Staubli VAL3: Sychron_points.dtx

public jointRx jJointRx[1000]
  [0] = {j1=4.067745, j2=-15.879896, j3=110.159334, j4=0.000858, j5=81.483567, j6=22.610962}
  [1] = {j1=4.051625, j2=-15.882186, j3=110.160996, j4=0.002059, j5=81.484196, j6=22.594711}
  [2] = {j1=4.035504, j2=-15.884473, j3=110.162655, j4=0.00326, j5=81.484824, j6=22.578459}
  [3] = {j1=4.019382, j2=-15.886755, j3=110.164311, j4=0.004461, j5=81.485452, j6=22.562206}
  [4] = {j1=4.003258, j2=-15.889034, j3=110.165965, j4=0.005663, j5=81.486079, j6=22.545952}
  [5] = {j1=3.987134, j2=-15.89131, j3=110.167615, j4=0.006864, j5=81.486705, j6=22.529696}
  [6] = {j1=3.971008, j2=-15.893581, j3=110.169263, j4=0.008065, j5=81.487331, j6=22.51344}
  [7] = {j1=3.954882, j2=-15.895849, j3=110.170908, j4=0.009267, j5=81.487956, j6=22.497183}
  [8] = {j1=3.938754, j2=-15.898113, j3=110.17255, j4=0.010468, j5=81.48858, j6=22.480924}
  [9] = {j1=3.922625, j2=-15.900374, j3=110.17419, j4=0.01167, j5=81.489204, j6=22.464665}
  [10] = {j1=3.906496, j2=-15.90263, j3=110.175826, j4=0.012872, j5=81.489828, j6=22.448405}
  [11] = {j1=3.890365, j2=-15.904883, j3=110.17746, j4=0.014073, j5=81.49045, j6=22.432143}
  [12] = {j1=3.874233, j2=-15.907132, j3=110.179091, j4=0.015275, j5=81.491073, j6=22.415881}
  [13] = {j1=3.8581, j2=-15.909377, j3=110.180719, j4=0.016477, j5=81.491694, j6=22.399617}
  [14] = {j1=3.841966, j2=-15.911619, j3=110.182345, j4=0.017679, j5=81.492315, j6=22.383352}
  [15] = {j1=3.825831, j2=-15.913857, j3=110.183967, j4=0.018881, j5=81.492935, j6=22.367087}
  [16] = {j1=3.809695, j2=-15.916091, j3=110.185587, j4=0.020083, j5=81.493555, j6=22.35082}
  [17] = {j1=3.793558, j2=-15.918321, j3=110.187204, j4=0.021286, j5=81.494174, j6=22.334552}
  [18] = {j1=3.77742, j2=-15.920548, j3=110.188818, j4=0.022488, j5=81.494792, j6=22.318284}
  [19] = {j1=3.76128, j2=-15.922771, j3=110.190429, j4=0.02369, j5=81.49541, j6=22.302014}
  [20] = {j1=3.74514, j2=-15.92499, j3=110.192038, j4=0.024893, j5=81.496028, j6=22.285743}
  [21] = {j1=3.728999, j2=-15.927205, j3=110.193644, j4=0.026095, j5=81.496644, j6=22.269472}
  [22] = {j1=3.712857, j2=-15.929416, j3=110.195247, j4=0.027298, j5=81.49726, j6=22.253199}
  [23] = {j1=3.696713, j2=-15.931624, j3=110.196847, j4=0.028501, j5=81.497876, j6=22.236925}
  [24] = {j1=3.680569, j2=-15.933828, j3=110.198444, j4=0.029703, j5=81.49849, j6=22.22065}
  [25] = {j1=3.664424, j2=-15.936029, j3=110.200039, j4=0.030906, j5=81.499105, j6=22.204374}
  [26] = {j1=3.648277, j2=-15.938225, j3=110.20163, j4=0.032109, j5=81.499718, j6=22.188098}
  [27] = {j1=3.63213, j2=-15.940418, j3=110.203219, j4=0.033312, j5=81.500331, j6=22.17182}
  [28] = {j1=3.615981, j2=-15.942607, j3=110.204805, j4=0.034515, j5=81.500943, j6=22.155541}
  [29] = {j1=3.599832, j2=-15.944792, j3=110.206389, j4=0.035718, j5=81.501555, j6=22.139261}
  [30] = {j1=3.583681, j2=-15.946974, j3=110.207969, j4=0.036921, j5=81.502166, j6=22.12298}
  [31] = {j1=3.56753, j2=-15.949151, j3=110.209547, j4=0.038124, j5=81.502777, j6=22.106699}
  [32] = {j1=3.551377, j2=-15.951325, j3=110.211122, j4=0.039328, j5=81.503386, j6=22.090416}
  [33] = {j1=3.535224, j2=-15.953496, j3=110.212694, j4=0.040531, j5=81.503996, j6=22.074132}
  [34] = {j1=3.51907, j2=-15.955662, j3=110.214263, j4=0.041734, j5=81.504604, j6=22.057847}
  [35] = {j1=3.502914, j2=-15.957825, j3=110.21583, j4=0.042938, j5=81.505212, j6=22.041562}
  [36] = {j1=3.486758, j2=-15.959984, j3=110.217393, j4=0.044141, j5=81.50582, j6=22.025275}
  [37] = {j1=3.4706, j2=-15.962139, j3=110.218954, j4=0.045345, j5=81.506426, j6=22.008987}
  [38] = {j1=3.454442, j2=-15.96429, j3=110.220512, j4=0.046549, j5=81.507032, j6=21.992699}
  [39] = {j1=3.438282, j2=-15.966438, j3=110.222068, j4=0.047752, j5=81.507638, j6=21.976409}
  [40] = {j1=3.422122, j2=-15.968582, j3=110.22362, j4=0.048956, j5=81.508243, j6=21.960119}
  [41] = {j1=3.40596, j2=-15.970722, j3=110.22517, j4=0.05016, j5=81.508847, j6=21.943827}
  [42] = {j1=3.389798, j2=-15.972858, j3=110.226717, j4=0.051364, j5=81.509451, j6=21.927534}
  [43] = {j1=3.373635, j2=-15.97499, j3=110.228261, j4=0.052568, j5=81.510054, j6=21.911241}
  [44] = {j1=3.35747, j2=-15.977119, j3=110.229802, j4=0.053772, j5=81.510656, j6=21.894947}
  [45] = {j1=3.341305, j2=-15.979244, j3=110.23134, j4=0.054976, j5=81.511258, j6=21.878651}
  [46] = {j1=3.325139, j2=-15.981365, j3=110.232876, j4=0.056181, j5=81.511859, j6=21.862355}
  [47] = {j1=3.308971, j2=-15.983483, j3=110.234409, j4=0.057385, j5=81.512459, j6=21.846058}
  [48] = {j1=3.292803, j2=-15.985597, j3=110.235939, j4=0.058589, j5=81.513059, j6=21.829759}
  [49] = {j1=3.276634, j2=-15.987706, j3=110.237466, j4=0.059794, j5=81.513659, j6=21.81346}
  [50] = {j1=3.260464, j2=-15.989813, j3=110.23899, j4=0.060998, j5=81.514257, j6=21.79716}
  [51] = {j1=3.244293, j2=-15.991915, j3=110.240512, j4=0.062203, j5=81.514855, j6=21.780859}
  [52] = {j1=3.228121, j2=-15.994014, j3=110.242031, j4=0.063407, j5=81.515452, j6=21.764557}
  [53] = {j1=3.211948, j2=-15.996108, j3=110.243547, j4=0.064612, j5=81.516049, j6=21.748254}
  [54] = {j1=3.195774, j2=-15.998199, j3=110.24506, j4=0.065816, j5=81.516645, j6=21.73195}
  [55] = {j1=3.179599, j2=-16.000287, j3=110.24657, j4=0.067021, j5=81.517241, j6=21.715645}
  [56] = {j1=3.163423, j2=-16.00237, j3=110.248078, j4=0.068226, j5=81.517836, j6=21.699339}
  [57] = {j1=3.147246, j2=-16.00445, j3=110.249583, j4=0.069431, j5=81.51843, j6=21.683033}
  [58] = {j1=3.131068, j2=-16.006526, j3=110.251085, j4=0.070636, j5=81.519023, j6=21.666725}
  [59] = {j1=3.11489, j2=-16.008598, j3=110.252584, j4=0.071841, j5=81.519616, j6=21.650417}
  [60] = {j1=3.09871, j2=-16.010666, j3=110.25408, j4=0.073046, j5=81.520209, j6=21.634107}
  [61] = {j1=3.082529, j2=-16.012731, j3=110.255574, j4=0.074251, j5=81.5208, j6=21.617797}
  [62] = {j1=3.066348, j2=-16.014792, j3=110.257064, j4=0.075456, j5=81.521391, j6=21.601485}
  [63] = {j1=3.050165, j2=-16.016849, j3=110.258552, j4=0.076662, j5=81.521982, j6=21.585173}
  [64] = {j1=3.033982, j2=-16.018902, j3=110.260037, j4=0.077867, j5=81.522572, j6=21.56886}
  [65] = {j1=3.017798, j2=-16.020951, j3=110.26152, j4=0.079072, j5=81.523161, j6=21.552546}
  [66] = {j1=3.001613, j2=-16.022997, j3=110.262999, j4=0.080278, j5=81.523749, j6=21.536231}
  [67] = {j1=2.985426, j2=-16.025039, j3=110.264476, j4=0.081483, j5=81.524337, j6=21.519915}
  [68] = {j1=2.969239, j2=-16.027077, j3=110.26595, j4=0.082689, j5=81.524924, j6=21.503599}
  [69] = {j1=2.953051, j2=-16.029111, j3=110.267421, j4=0.083894, j5=81.525511, j6=21.487281}
  [70] = {j1=2.936863, j2=-16.031142, j3=110.268889, j4=0.0851, j5=81.526097, j6=21.470962}
  [71] = {j1=2.920673, j2=-16.033169, j3=110.270355, j4=0.086306, j5=81.526682, j6=21.454643}
  [72] = {j1=2.904482, j2=-16.035192, j3=110.271817, j4=0.087512, j5=81.527267, j6=21.438323}
  [73] = {j1=2.88829, j2=-16.037211, j3=110.273277, j4=0.088718, j5=81.527851, j6=21.422001}
  [74] = {j1=2.872098, j2=-16.039226, j3=110.274734, j4=0.089923, j5=81.528434, j6=21.405679}
  [75] = {j1=2.855905, j2=-16.041238, j3=110.276189, j4=0.091129, j5=81.529017, j6=21.389356}
  [76] = {j1=2.83971, j2=-16.043246, j3=110.27764, j4=0.092335, j5=81.529599, j6=21.373033}
  [77] = {j1=2.823515, j2=-16.04525, j3=110.279089, j4=0.093541, j5=81.53018, j6=21.356708}
  [78] = {j1=2.807319, j2=-16.04725, j3=110.280535, j4=0.094748, j5=81.530761, j6=21.340382}
  [79] = {j1=2.791122, j2=-16.049246, j3=110.281978, j4=0.095954, j5=81.531341, j6=21.324056}
  [80] = {j1=2.774924, j2=-16.051239, j3=110.283418, j4=0.09716, j5=81.531921, j6=21.307728}
  [81] = {j1=2.758725, j2=-16.053228, j3=110.284855, j4=0.098366, j5=81.5325, j6=21.2914}
  [82] = {j1=2.742526, j2=-16.055213, j3=110.28629, j4=0.099573, j5=81.533078, j6=21.275071}
  [83] = {j1=2.726325, j2=-16.057194, j3=110.287722, j4=0.100779, j5=81.533656, j6=21.258741}
  [84] = {j1=2.710124, j2=-16.059172, j3=110.289151, j4=0.101985, j5=81.534233, j6=21.24241}
  [85] = {j1=2.693922, j2=-16.061146, j3=110.290577, j4=0.103192, j5=81.534809, j6=21.226079}
  [86] = {j1=2.677718, j2=-16.063115, j3=110.292, j4=0.104399, j5=81.535385, j6=21.209746}
  [87] = {j1=2.661514, j2=-16.065082, j3=110.293421, j4=0.105605, j5=81.53596, j6=21.193413}
  [88] = {j1=2.645309, j2=-16.067044, j3=110.294839, j4=0.106812, j5=81.536534, j6=21.177078}
  [89] = {j1=2.629104, j2=-16.069002, j3=110.296253, j4=0.108019, j5=81.537108, j6=21.160743}
  [90] = {j1=2.612897, j2=-16.070957, j3=110.297666, j4=0.109225, j5=81.537681, j6=21.144407}
  [91] = {j1=2.59669, j2=-16.072908, j3=110.299075, j4=0.110432, j5=81.538253, j6=21.128071}
  [92] = {j1=2.580481, j2=-16.074855, j3=110.300481, j4=0.111639, j5=81.538825, j6=21.111733}
  [93] = {j1=2.564272, j2=-16.076798, j3=110.301885, j4=0.112846, j5=81.539396, j6=21.095394}
  [94] = {j1=2.548062, j2=-16.078738, j3=110.303286, j4=0.114053, j5=81.539967, j6=21.079055}
  [95] = {j1=2.531851, j2=-16.080674, j3=110.304684, j4=0.11526, j5=81.540537, j6=21.062715}
  [96] = {j1=2.515639, j2=-16.082606, j3=110.30608, j4=0.116467, j5=81.541106, j6=21.046374}
  [97] = {j1=2.499427, j2=-16.084534, j3=110.307472, j4=0.117674, j5=81.541674, j6=21.030032}
  [98] = {j1=2.483213, j2=-16.086458, j3=110.308862, j4=0.118881, j5=81.542242, j6=21.01369}
  [99] = {j1=2.466999, j2=-16.088378, j3=110.310249, j4=0.120089, j5=81.542809, j6=20.997346}
  [100] = {j1=2.450784, j2=-16.090295, j3=110.311633, j4=0.121296, j5=81.543376, j6=20.981002}
  [101] = {j1=2.434568, j2=-16.092208, j3=110.313014, j4=0.122503, j5=81.543942, j6=20.964657}
  [102] = {j1=2.418351, j2=-16.094117, j3=110.314392, j4=0.123711, j5=81.544507, j6=20.948311}
  [103] = {j1=2.402134, j2=-16.096023, j3=110.315768, j4=0.124918, j5=81.545072, j6=20.931964}
  [104] = {j1=2.385915, j2=-16.097924, j3=110.317141, j4=0.126126, j5=81.545636, j6=20.915617}
  [105] = {j1=2.369696, j2=-16.099822, j3=110.318511, j4=0.127333, j5=81.546199, j6=20.899268}
  [106] = {j1=2.353476, j2=-16.101716, j3=110.319878, j4=0.128541, j5=81.546762, j6=20.882919}
  [107] = {j1=2.337255, j2=-16.103606, j3=110.321243, j4=0.129748, j5=81.547324, j6=20.866569}
  [108] = {j1=2.321033, j2=-16.105492, j3=110.322604, j4=0.130956, j5=81.547885, j6=20.850218}
  [109] = {j1=2.304811, j2=-16.107374, j3=110.323963, j4=0.132164, j5=81.548446, j6=20.833867}
  [110] = {j1=2.288587, j2=-16.109253, j3=110.325319, j4=0.133371, j5=81.549006, j6=20.817514}
  [111] = {j1=2.272363, j2=-16.111128, j3=110.326672, j4=0.134579, j5=81.549565, j6=20.801161}
  [112] = {j1=2.256138, j2=-16.112999, j3=110.328023, j4=0.135787, j5=81.550124, j6=20.784807}
  [113] = {j1=2.239912, j2=-16.114866, j3=110.32937, j4=0.136995, j5=81.550682, j6=20.768453}
  [114] = {j1=2.223686, j2=-16.11673, j3=110.330715, j4=0.138203, j5=81.551239, j6=20.752097}
  [115] = {j1=2.207459, j2=-16.118589, j3=110.332057, j4=0.139411, j5=81.551796, j6=20.735741}
  [116] = {j1=2.19123, j2=-16.120445, j3=110.333396, j4=0.140619, j5=81.552352, j6=20.719384}
  [117] = {j1=2.175001, j2=-16.122297, j3=110.334732, j4=0.141827, j5=81.552907, j6=20.703026}
  [118] = {j1=2.158772, j2=-16.124145, j3=110.336066, j4=0.143035, j5=81.553462, j6=20.686667}
  [119] = {j1=2.142541, j2=-16.125989, j3=110.337397, j4=0.144243, j5=81.554016, j6=20.670308}
  [120] = {j1=2.12631, j2=-16.12783, j3=110.338725, j4=0.145452, j5=81.554569, j6=20.653948}
  [121] = {j1=2.110078, j2=-16.129667, j3=110.34005, j4=0.14666, j5=81.555122, j6=20.637587}
  [122] = {j1=2.093845, j2=-16.1315, j3=110.341372, j4=0.147868, j5=81.555674, j6=20.621225}
  [123] = {j1=2.077611, j2=-16.133329, j3=110.342692, j4=0.149076, j5=81.556226, j6=20.604862}
  [124] = {j1=2.061376, j2=-16.135154, j3=110.344008, j4=0.150285, j5=81.556776, j6=20.588499}
  [125] = {j1=2.045141, j2=-16.136975, j3=110.345322, j4=0.151493, j5=81.557327, j6=20.572135}
  [126] = {j1=2.028905, j2=-16.138793, j3=110.346633, j4=0.152702, j5=81.557876, j6=20.55577}
  [127] = {j1=2.012668, j2=-16.140607, j3=110.347941, j4=0.15391, j5=81.558425, j6=20.539405}
  [128] = {j1=1.996431, j2=-16.142417, j3=110.349247, j4=0.155119, j5=81.558973, j6=20.523038}
  [129] = {j1=1.980192, j2=-16.144223, j3=110.350549, j4=0.156327, j5=81.55952, j6=20.506671}
  [130] = {j1=1.963953, j2=-16.146026, j3=110.351849, j4=0.157536, j5=81.560067, j6=20.490304}
  [131] = {j1=1.947714, j2=-16.147824, j3=110.353146, j4=0.158745, j5=81.560613, j6=20.473935}
  [132] = {j1=1.931473, j2=-16.149619, j3=110.354441, j4=0.159954, j5=81.561159, j6=20.457566}
  [133] = {j1=1.915232, j2=-16.15141, j3=110.355732, j4=0.161162, j5=81.561703, j6=20.441196}
  [134] = {j1=1.898989, j2=-16.153197, j3=110.357021, j4=0.162371, j5=81.562247, j6=20.424825}
  [135] = {j1=1.882747, j2=-16.15498, j3=110.358306, j4=0.16358, j5=81.562791, j6=20.408454}
  [136] = {j1=1.866503, j2=-16.15676, j3=110.359589, j4=0.164789, j5=81.563334, j6=20.392081}
  [137] = {j1=1.850259, j2=-16.158535, j3=110.360869, j4=0.165998, j5=81.563876, j6=20.375708}
  [138] = {j1=1.834014, j2=-16.160307, j3=110.362147, j4=0.167207, j5=81.564417, j6=20.359335}
  [139] = {j1=1.817768, j2=-16.162075, j3=110.363421, j4=0.168416, j5=81.564958, j6=20.34296}
  [140] = {j1=1.801521, j2=-16.163839, j3=110.364693, j4=0.169625, j5=81.565498, j6=20.326585}
  [141] = {j1=1.785274, j2=-16.165599, j3=110.365962, j4=0.170834, j5=81.566037, j6=20.310209}
  [142] = {j1=1.769026, j2=-16.167356, j3=110.367228, j4=0.172043, j5=81.566576, j6=20.293833}
  [143] = {j1=1.752777, j2=-16.169109, j3=110.368492, j4=0.173252, j5=81.567114, j6=20.277455}
  [144] = {j1=1.736527, j2=-16.170857, j3=110.369752, j4=0.174461, j5=81.567651, j6=20.261077}
  [145] = {j1=1.720277, j2=-16.172602, j3=110.37101, j4=0.175671, j5=81.568188, j6=20.244699}
  [146] = {j1=1.704026, j2=-16.174344, j3=110.372265, j4=0.17688, j5=81.568724, j6=20.228319}
  [147] = {j1=1.687775, j2=-16.176081, j3=110.373517, j4=0.178089, j5=81.569259, j6=20.211939}
  [148] = {j1=1.671522, j2=-16.177815, j3=110.374766, j4=0.179298, j5=81.569794, j6=20.195558}
  [149] = {j1=1.655269, j2=-16.179544, j3=110.376012, j4=0.180508, j5=81.570328, j6=20.179177}
  [150] = {j1=1.639015, j2=-16.18127, j3=110.377256, j4=0.181717, j5=81.570861, j6=20.162795}
  [151] = {j1=1.622761, j2=-16.182992, j3=110.378497, j4=0.182927, j5=81.571394, j6=20.146412}
  [152] = {j1=1.606505, j2=-16.18471, j3=110.379735, j4=0.184136, j5=81.571926, j6=20.130028}
  [153] = {j1=1.59025, j2=-16.186425, j3=110.38097, j4=0.185346, j5=81.572457, j6=20.113644}
  [154] = {j1=1.573993, j2=-16.188135, j3=110.382203, j4=0.186555, j5=81.572988, j6=20.097259}
  [155] = {j1=1.557736, j2=-16.189842, j3=110.383432, j4=0.187765, j5=81.573518, j6=20.080873}
  [156] = {j1=1.541478, j2=-16.191545, j3=110.384659, j4=0.188974, j5=81.574047, j6=20.064487}
  [157] = {j1=1.525219, j2=-16.193244, j3=110.385883, j4=0.190184, j5=81.574576, j6=20.0481}
  [158] = {j1=1.508959, j2=-16.194939, j3=110.387104, j4=0.191394, j5=81.575104, j6=20.031712}
  [159] = {j1=1.492699, j2=-16.196631, j3=110.388322, j4=0.192603, j5=81.575631, j6=20.015324}
  [160] = {j1=1.476438, j2=-16.198318, j3=110.389538, j4=0.193813, j5=81.576157, j6=19.998935}
  [161] = {j1=1.460177, j2=-16.200002, j3=110.390751, j4=0.195023, j5=81.576683, j6=19.982545}
  [162] = {j1=1.443915, j2=-16.201682, j3=110.391961, j4=0.196233, j5=81.577209, j6=19.966155}
  [163] = {j1=1.427652, j2=-16.203358, j3=110.393168, j4=0.197443, j5=81.577733, j6=19.949764}
  [164] = {j1=1.411388, j2=-16.20503, j3=110.394372, j4=0.198653, j5=81.578257, j6=19.933372}
  [165] = {j1=1.395124, j2=-16.206698, j3=110.395574, j4=0.199862, j5=81.57878, j6=19.91698}
  [166] = {j1=1.378859, j2=-16.208363, j3=110.396772, j4=0.201072, j5=81.579302, j6=19.900586}
  [167] = {j1=1.362594, j2=-16.210024, j3=110.397968, j4=0.202282, j5=81.579824, j6=19.884193}
  [168] = {j1=1.346328, j2=-16.211681, j3=110.399161, j4=0.203492, j5=81.580345, j6=19.867798}
  [169] = {j1=1.330061, j2=-16.213334, j3=110.400352, j4=0.204702, j5=81.580866, j6=19.851403}
  [170] = {j1=1.313793, j2=-16.214983, j3=110.401539, j4=0.205912, j5=81.581385, j6=19.835008}
  [171] = {j1=1.297525, j2=-16.216628, j3=110.402724, j4=0.207123, j5=81.581904, j6=19.818612}
  [172] = {j1=1.281256, j2=-16.21827, j3=110.403905, j4=0.208333, j5=81.582423, j6=19.802215}
  [173] = {j1=1.264987, j2=-16.219907, j3=110.405085, j4=0.209543, j5=81.58294, j6=19.785817}
  [174] = {j1=1.248717, j2=-16.221541, j3=110.406261, j4=0.210753, j5=81.583457, j6=19.769419}
  [175] = {j1=1.232446, j2=-16.223171, j3=110.407434, j4=0.211963, j5=81.583974, j6=19.75302}
  [176] = {j1=1.216174, j2=-16.224797, j3=110.408605, j4=0.213173, j5=81.584489, j6=19.736621}
  [177] = {j1=1.199902, j2=-16.22642, j3=110.409772, j4=0.214384, j5=81.585004, j6=19.720221}
  [178] = {j1=1.183629, j2=-16.228038, j3=110.410937, j4=0.215594, j5=81.585518, j6=19.70382}
  [179] = {j1=1.167356, j2=-16.229653, j3=110.4121, j4=0.216804, j5=81.586032, j6=19.687418}
  [180] = {j1=1.151082, j2=-16.231263, j3=110.413259, j4=0.218015, j5=81.586545, j6=19.671017}
  [181] = {j1=1.134807, j2=-16.23287, j3=110.414416, j4=0.219225, j5=81.587057, j6=19.654614}
  [182] = {j1=1.118532, j2=-16.234473, j3=110.415569, j4=0.220435, j5=81.587568, j6=19.638211}
  [183] = {j1=1.102256, j2=-16.236073, j3=110.41672, j4=0.221646, j5=81.588079, j6=19.621807}
  [184] = {j1=1.08598, j2=-16.237668, j3=110.417868, j4=0.222856, j5=81.588589, j6=19.605402}
  [185] = {j1=1.069703, j2=-16.23926, j3=110.419014, j4=0.224067, j5=81.589099, j6=19.588997}
  [186] = {j1=1.053425, j2=-16.240847, j3=110.420156, j4=0.225277, j5=81.589607, j6=19.572592}
  [187] = {j1=1.037147, j2=-16.242431, j3=110.421296, j4=0.226488, j5=81.590115, j6=19.556186}
  [188] = {j1=1.020868, j2=-16.244011, j3=110.422433, j4=0.227698, j5=81.590623, j6=19.539779}
  [189] = {j1=1.004588, j2=-16.245587, j3=110.423567, j4=0.228909, j5=81.591129, j6=19.523371}
  [190] = {j1=0.988308, j2=-16.247159, j3=110.424698, j4=0.23012, j5=81.591635, j6=19.506963}
  [191] = {j1=0.972027, j2=-16.248728, j3=110.425826, j4=0.23133, j5=81.592141, j6=19.490555}
  [192] = {j1=0.955745, j2=-16.250292, j3=110.426952, j4=0.232541, j5=81.592645, j6=19.474145}
  [193] = {j1=0.939463, j2=-16.251853, j3=110.428075, j4=0.233752, j5=81.593149, j6=19.457736}
  [194] = {j1=0.923181, j2=-16.25341, j3=110.429195, j4=0.234962, j5=81.593652, j6=19.441325}
  [195] = {j1=0.906898, j2=-16.254963, j3=110.430312, j4=0.236173, j5=81.594155, j6=19.424914}
  [196] = {j1=0.890614, j2=-16.256512, j3=110.431426, j4=0.237384, j5=81.594656, j6=19.408503}
  [197] = {j1=0.874329, j2=-16.258058, j3=110.432538, j4=0.238594, j5=81.595157, j6=19.392091}
  [198] = {j1=0.858044, j2=-16.259599, j3=110.433647, j4=0.239805, j5=81.595658, j6=19.375678}
  [199] = {j1=0.841759, j2=-16.261137, j3=110.434753, j4=0.241016, j5=81.596157, j6=19.359265}
  [200] = {j1=0.825473, j2=-16.262671, j3=110.435856, j4=0.242227, j5=81.596656, j6=19.342851}
  [201] = {j1=0.809186, j2=-16.264201, j3=110.436956, j4=0.243438, j5=81.597155, j6=19.326436}
  [202] = {j1=0.792898, j2=-16.265727, j3=110.438054, j4=0.244649, j5=81.597652, j6=19.310021}
  [203] = {j1=0.77661, j2=-16.267249, j3=110.439148, j4=0.24586, j5=81.598149, j6=19.293606}
  [204] = {j1=0.760322, j2=-16.268767, j3=110.44024, j4=0.24707, j5=81.598645, j6=19.27719}
  [205] = {j1=0.744033, j2=-16.270282, j3=110.441329, j4=0.248281, j5=81.599141, j6=19.260773}
  [206] = {j1=0.727743, j2=-16.271792, j3=110.442415, j4=0.249492, j5=81.599636, j6=19.244356}
  [207] = {j1=0.711453, j2=-16.273299, j3=110.443499, j4=0.250703, j5=81.60013, j6=19.227938}
  [208] = {j1=0.695162, j2=-16.274802, j3=110.44458, j4=0.251914, j5=81.600623, j6=19.21152}
  [209] = {j1=0.678871, j2=-16.276301, j3=110.445657, j4=0.253125, j5=81.601116, j6=19.195101}
  [210] = {j1=0.662579, j2=-16.277796, j3=110.446732, j4=0.254336, j5=81.601608, j6=19.178681}
  [211] = {j1=0.646287, j2=-16.279288, j3=110.447805, j4=0.255547, j5=81.602099, j6=19.162261}
  [212] = {j1=0.629994, j2=-16.280775, j3=110.448874, j4=0.256758, j5=81.60259, j6=19.145841}
  [213] = {j1=0.6137, j2=-16.282259, j3=110.449941, j4=0.25797, j5=81.60308, j6=19.12942}
  [214] = {j1=0.597406, j2=-16.283739, j3=110.451004, j4=0.259181, j5=81.603569, j6=19.112998}
  [215] = {j1=0.581111, j2=-16.285214, j3=110.452065, j4=0.260392, j5=81.604057, j6=19.096576}
  [216] = {j1=0.564816, j2=-16.286687, j3=110.453123, j4=0.261603, j5=81.604545, j6=19.080153}
  [217] = {j1=0.548521, j2=-16.288155, j3=110.454179, j4=0.262814, j5=81.605032, j6=19.06373}
  [218] = {j1=0.532224, j2=-16.289619, j3=110.455231, j4=0.264025, j5=81.605518, j6=19.047307}
  [219] = {j1=0.515928, j2=-16.29108, j3=110.456281, j4=0.265236, j5=81.606004, j6=19.030882}
  [220] = {j1=0.49963, j2=-16.292536, j3=110.457328, j4=0.266448, j5=81.606489, j6=19.014458}
  [221] = {j1=0.483332, j2=-16.293989, j3=110.458372, j4=0.267659, j5=81.606973, j6=18.998032}
  [222] = {j1=0.467034, j2=-16.295438, j3=110.459413, j4=0.26887, j5=81.607457, j6=18.981607}
  [223] = {j1=0.450735, j2=-16.296883, j3=110.460452, j4=0.270081, j5=81.60794, j6=18.96518}
  [224] = {j1=0.434436, j2=-16.298324, j3=110.461487, j4=0.271293, j5=81.608422, j6=18.948753}
  [225] = {j1=0.418136, j2=-16.299761, j3=110.46252, j4=0.272504, j5=81.608903, j6=18.932326}
  [226] = {j1=0.401835, j2=-16.301195, j3=110.46355, j4=0.273715, j5=81.609384, j6=18.915898}
  [227] = {j1=0.385534, j2=-16.302624, j3=110.464578, j4=0.274926, j5=81.609864, j6=18.89947}
  [228] = {j1=0.369233, j2=-16.30405, j3=110.465602, j4=0.276138, j5=81.610343, j6=18.883041}
  [229] = {j1=0.352931, j2=-16.305472, j3=110.466624, j4=0.277349, j5=81.610822, j6=18.866612}
  [230] = {j1=0.336628, j2=-16.30689, j3=110.467642, j4=0.27856, j5=81.6113, j6=18.850182}
  [231] = {j1=0.320325, j2=-16.308304, j3=110.468658, j4=0.279772, j5=81.611777, j6=18.833752}
  [232] = {j1=0.304022, j2=-16.309714, j3=110.469671, j4=0.280983, j5=81.612253, j6=18.817321}
  [233] = {j1=0.287718, j2=-16.31112, j3=110.470682, j4=0.282195, j5=81.612729, j6=18.80089}
  [234] = {j1=0.271413, j2=-16.312523, j3=110.471689, j4=0.283406, j5=81.613204, j6=18.784458}
  [235] = {j1=0.255108, j2=-16.313921, j3=110.472694, j4=0.284617, j5=81.613678, j6=18.768026}
  [236] = {j1=0.238803, j2=-16.315316, j3=110.473696, j4=0.285829, j5=81.614152, j6=18.751593}
  [237] = {j1=0.222497, j2=-16.316707, j3=110.474695, j4=0.28704, j5=81.614625, j6=18.73516}
  [238] = {j1=0.20619, j2=-16.318094, j3=110.475691, j4=0.288252, j5=81.615097, j6=18.718726}
  [239] = {j1=0.189883, j2=-16.319477, j3=110.476685, j4=0.289463, j5=81.615569, j6=18.702292}
  [240] = {j1=0.173576, j2=-16.320856, j3=110.477676, j4=0.290675, j5=81.616039, j6=18.685858}
  [241] = {j1=0.157268, j2=-16.322232, j3=110.478663, j4=0.291886, j5=81.61651, j6=18.669423}
  [242] = {j1=0.14096, j2=-16.323603, j3=110.479648, j4=0.293097, j5=81.616979, j6=18.652987}
  [243] = {j1=0.124651, j2=-16.324971, j3=110.480631, j4=0.294309, j5=81.617447, j6=18.636551}
  [244] = {j1=0.108341, j2=-16.326335, j3=110.48161, j4=0.29552, j5=81.617915, j6=18.620115}
  [245] = {j1=0.092032, j2=-16.327695, j3=110.482587, j4=0.296732, j5=81.618383, j6=18.603678}
  [246] = {j1=0.075721, j2=-16.329051, j3=110.48356, j4=0.297943, j5=81.618849, j6=18.587241}
  [247] = {j1=0.059411, j2=-16.330403, j3=110.484531, j4=0.299155, j5=81.619315, j6=18.570803}
  [248] = {j1=0.043099, j2=-16.331751, j3=110.4855, j4=0.300367, j5=81.61978, j6=18.554364}
  [249] = {j1=0.026788, j2=-16.333096, j3=110.486465, j4=0.301578, j5=81.620244, j6=18.537926}
  [250] = {j1=0.010476, j2=-16.334436, j3=110.487427, j4=0.30279, j5=81.620708, j6=18.521487}
  [251] = {j1=-0.005837, j2=-16.335773, j3=110.488387, j4=0.304001, j5=81.621171, j6=18.505047}
  [252] = {j1=-0.02215, j2=-16.337106, j3=110.489344, j4=0.305213, j5=81.621633, j6=18.488607}
  [253] = {j1=-0.038463, j2=-16.338434, j3=110.490298, j4=0.306424, j5=81.622094, j6=18.472167}
  [254] = {j1=-0.054777, j2=-16.339759, j3=110.491249, j4=0.307636, j5=81.622555, j6=18.455726}
  [255] = {j1=-0.071092, j2=-16.341081, j3=110.492198, j4=0.308847, j5=81.623015, j6=18.439284}
  [256] = {j1=-0.087406, j2=-16.342398, j3=110.493144, j4=0.310059, j5=81.623475, j6=18.422843}
  [257] = {j1=-0.103722, j2=-16.343711, j3=110.494086, j4=0.311271, j5=81.623933, j6=18.406401}
  [258] = {j1=-0.120037, j2=-16.345021, j3=110.495026, j4=0.312482, j5=81.624391, j6=18.389958}
  [259] = {j1=-0.136353, j2=-16.346326, j3=110.495964, j4=0.313694, j5=81.624848, j6=18.373515}
  [260] = {j1=-0.15267, j2=-16.347628, j3=110.496898, j4=0.314905, j5=81.625305, j6=18.357072}
  [261] = {j1=-0.168987, j2=-16.348926, j3=110.49783, j4=0.316117, j5=81.62576, j6=18.340628}
  [262] = {j1=-0.185304, j2=-16.35022, j3=110.498758, j4=0.317329, j5=81.626215, j6=18.324184}
  [263] = {j1=-0.201622, j2=-16.35151, j3=110.499684, j4=0.31854, j5=81.62667, j6=18.307739}
  [264] = {j1=-0.21794, j2=-16.352796, j3=110.500608, j4=0.319752, j5=81.627123, j6=18.291294}
  [265] = {j1=-0.234259, j2=-16.354079, j3=110.501528, j4=0.320963, j5=81.627576, j6=18.274848}
  [266] = {j1=-0.250578, j2=-16.355357, j3=110.502445, j4=0.322175, j5=81.628028, j6=18.258403}
  [267] = {j1=-0.266897, j2=-16.356632, j3=110.50336, j4=0.323387, j5=81.62848, j6=18.241956}
  [268] = {j1=-0.283217, j2=-16.357903, j3=110.504272, j4=0.324598, j5=81.62893, j6=18.22551}
  [269] = {j1=-0.299537, j2=-16.359169, j3=110.505181, j4=0.32581, j5=81.62938, j6=18.209063}
  [270] = {j1=-0.315858, j2=-16.360432, j3=110.506087, j4=0.327022, j5=81.629829, j6=18.192615}
  [271] = {j1=-0.332179, j2=-16.361691, j3=110.506991, j4=0.328233, j5=81.630278, j6=18.176167}
  [272] = {j1=-0.3485, j2=-16.362947, j3=110.507892, j4=0.329445, j5=81.630726, j6=18.159719}
  [273] = {j1=-0.364822, j2=-16.364198, j3=110.508789, j4=0.330656, j5=81.631173, j6=18.143271}
  [274] = {j1=-0.381144, j2=-16.365445, j3=110.509684, j4=0.331868, j5=81.631619, j6=18.126822}
  [275] = {j1=-0.397467, j2=-16.366689, j3=110.510577, j4=0.33308, j5=81.632065, j6=18.110372}
  [276] = {j1=-0.41379, j2=-16.367928, j3=110.511466, j4=0.334291, j5=81.632509, j6=18.093923}
  [277] = {j1=-0.430113, j2=-16.369164, j3=110.512353, j4=0.335503, j5=81.632954, j6=18.077472}
  [278] = {j1=-0.446437, j2=-16.370396, j3=110.513236, j4=0.336715, j5=81.633397, j6=18.061022}
  [279] = {j1=-0.462761, j2=-16.371624, j3=110.514117, j4=0.337926, j5=81.63384, j6=18.044571}
  [280] = {j1=-0.479086, j2=-16.372848, j3=110.514996, j4=0.339138, j5=81.634282, j6=18.02812}
  [281] = {j1=-0.495411, j2=-16.374068, j3=110.515871, j4=0.340349, j5=81.634723, j6=18.011668}
  [282] = {j1=-0.511736, j2=-16.375285, j3=110.516743, j4=0.341561, j5=81.635163, j6=17.995217}
  [283] = {j1=-0.528062, j2=-16.376497, j3=110.517613, j4=0.342773, j5=81.635603, j6=17.978764}
  [284] = {j1=-0.544388, j2=-16.377706, j3=110.51848, j4=0.343984, j5=81.636042, j6=17.962312}
  [285] = {j1=-0.560714, j2=-16.37891, j3=110.519344, j4=0.345196, j5=81.636481, j6=17.945859}
  [286] = {j1=-0.577041, j2=-16.380111, j3=110.520205, j4=0.346408, j5=81.636918, j6=17.929405}
  [287] = {j1=-0.593368, j2=-16.381308, j3=110.521064, j4=0.347619, j5=81.637355, j6=17.912952}
  [288] = {j1=-0.609695, j2=-16.382501, j3=110.521919, j4=0.348831, j5=81.637791, j6=17.896498}
  [289] = {j1=-0.626023, j2=-16.38369, j3=110.522772, j4=0.350042, j5=81.638227, j6=17.880043}
  [290] = {j1=-0.642351, j2=-16.384875, j3=110.523622, j4=0.351254, j5=81.638661, j6=17.863589}
  [291] = {j1=-0.65868, j2=-16.386057, j3=110.524469, j4=0.352466, j5=81.639095, j6=17.847134}
  [292] = {j1=-0.675008, j2=-16.387234, j3=110.525314, j4=0.353677, j5=81.639528, j6=17.830678}
  [293] = {j1=-0.691338, j2=-16.388408, j3=110.526155, j4=0.354889, j5=81.639961, j6=17.814222}
  [294] = {j1=-0.707667, j2=-16.389577, j3=110.526994, j4=0.3561, j5=81.640393, j6=17.797766}
  [295] = {j1=-0.723997, j2=-16.390743, j3=110.52783, j4=0.357312, j5=81.640824, j6=17.78131}
  [296] = {j1=-0.740327, j2=-16.391905, j3=110.528663, j4=0.358523, j5=81.641254, j6=17.764853}
  [297] = {j1=-0.756658, j2=-16.393063, j3=110.529494, j4=0.359735, j5=81.641683, j6=17.748396}
  [298] = {j1=-0.772989, j2=-16.394217, j3=110.530321, j4=0.360947, j5=81.642112, j6=17.731939}
  [299] = {j1=-0.78932, j2=-16.395367, j3=110.531146, j4=0.362158, j5=81.64254, j6=17.715481}
  [300] = {j1=-0.805651, j2=-16.396513, j3=110.531968, j4=0.36337, j5=81.642968, j6=17.699023}
  [301] = {j1=-0.821983, j2=-16.397656, j3=110.532787, j4=0.364581, j5=81.643394, j6=17.682565}
  [302] = {j1=-0.838315, j2=-16.398794, j3=110.533603, j4=0.365793, j5=81.64382, j6=17.666107}
  [303] = {j1=-0.854648, j2=-16.399929, j3=110.534416, j4=0.367004, j5=81.644245, j6=17.649648}
  [304] = {j1=-0.87098, j2=-16.401059, j3=110.535227, j4=0.368216, j5=81.64467, j6=17.633189}
  [305] = {j1=-0.887314, j2=-16.402186, j3=110.536035, j4=0.369427, j5=81.645093, j6=17.616729}
  [306] = {j1=-0.903647, j2=-16.403309, j3=110.53684, j4=0.370639, j5=81.645516, j6=17.600269}
  [307] = {j1=-0.919981, j2=-16.404428, j3=110.537642, j4=0.37185, j5=81.645939, j6=17.583809}
  [308] = {j1=-0.936315, j2=-16.405543, j3=110.538441, j4=0.373062, j5=81.64636, j6=17.567349}
  [309] = {j1=-0.952649, j2=-16.406655, j3=110.539238, j4=0.374273, j5=81.646781, j6=17.550888}
  [310] = {j1=-0.968984, j2=-16.407762, j3=110.540032, j4=0.375485, j5=81.647201, j6=17.534427}
  [311] = {j1=-0.985318, j2=-16.408865, j3=110.540822, j4=0.376696, j5=81.64762, j6=17.517966}
  [312] = {j1=-1.001654, j2=-16.409965, j3=110.541611, j4=0.377907, j5=81.648039, j6=17.501505}
  [313] = {j1=-1.017989, j2=-16.41106, j3=110.542396, j4=0.379119, j5=81.648456, j6=17.485043}
  [314] = {j1=-1.034325, j2=-16.412152, j3=110.543178, j4=0.38033, j5=81.648873, j6=17.468581}
  [315] = {j1=-1.050661, j2=-16.41324, j3=110.543958, j4=0.381542, j5=81.64929, j6=17.452119}
  [316] = {j1=-1.066997, j2=-16.414324, j3=110.544735, j4=0.382753, j5=81.649705, j6=17.435656}
  [317] = {j1=-1.083334, j2=-16.415404, j3=110.545509, j4=0.383964, j5=81.65012, j6=17.419193}
  [318] = {j1=-1.099671, j2=-16.41648, j3=110.54628, j4=0.385176, j5=81.650534, j6=17.40273}
  [319] = {j1=-1.116008, j2=-16.417552, j3=110.547048, j4=0.386387, j5=81.650948, j6=17.386267}
  [320] = {j1=-1.132345, j2=-16.418621, j3=110.547814, j4=0.387598, j5=81.65136, j6=17.369803}
  [321] = {j1=-1.148683, j2=-16.419685, j3=110.548577, j4=0.38881, j5=81.651772, j6=17.353339}
  [322] = {j1=-1.165021, j2=-16.420746, j3=110.549337, j4=0.390021, j5=81.652183, j6=17.336875}
  [323] = {j1=-1.181359, j2=-16.421802, j3=110.550094, j4=0.391232, j5=81.652594, j6=17.32041}
  [324] = {j1=-1.197698, j2=-16.422855, j3=110.550848, j4=0.392444, j5=81.653003, j6=17.303946}
  [325] = {j1=-1.214036, j2=-16.423904, j3=110.5516, j4=0.393655, j5=81.653412, j6=17.287481}
  [326] = {j1=-1.230375, j2=-16.424949, j3=110.552348, j4=0.394866, j5=81.65382, j6=17.271016}
  [327] = {j1=-1.246715, j2=-16.42599, j3=110.553094, j4=0.396077, j5=81.654228, j6=17.25455}
  [328] = {j1=-1.263054, j2=-16.427027, j3=110.553837, j4=0.397289, j5=81.654634, j6=17.238085}
  [329] = {j1=-1.279394, j2=-16.42806, j3=110.554578, j4=0.3985, j5=81.65504, j6=17.221619}
  [330] = {j1=-1.295734, j2=-16.429089, j3=110.555315, j4=0.399711, j5=81.655445, j6=17.205153}
  [331] = {j1=-1.312074, j2=-16.430115, j3=110.55605, j4=0.400922, j5=81.65585, j6=17.188686}
  [332] = {j1=-1.328415, j2=-16.431136, j3=110.556782, j4=0.402133, j5=81.656254, j6=17.17222}
  [333] = {j1=-1.344755, j2=-16.432154, j3=110.557511, j4=0.403344, j5=81.656657, j6=17.155753}
  [334] = {j1=-1.361096, j2=-16.433168, j3=110.558237, j4=0.404556, j5=81.657059, j6=17.139286}
  [335] = {j1=-1.377437, j2=-16.434177, j3=110.55896, j4=0.405767, j5=81.65746, j6=17.122819}
  [336] = {j1=-1.393779, j2=-16.435183, j3=110.559681, j4=0.406978, j5=81.657861, j6=17.106351}
  [337] = {j1=-1.41012, j2=-16.436185, j3=110.560398, j4=0.408189, j5=81.658261, j6=17.089883}
  [338] = {j1=-1.426462, j2=-16.437183, j3=110.561113, j4=0.4094, j5=81.65866, j6=17.073416}
  [339] = {j1=-1.442804, j2=-16.438178, j3=110.561825, j4=0.410611, j5=81.659059, j6=17.056947}
  [340] = {j1=-1.459147, j2=-16.439168, j3=110.562535, j4=0.411822, j5=81.659456, j6=17.040479}
  [341] = {j1=-1.475489, j2=-16.440154, j3=110.563241, j4=0.413033, j5=81.659853, j6=17.024011}
  [342] = {j1=-1.491832, j2=-16.441137, j3=110.563945, j4=0.414244, j5=81.66025, j6=17.007542}
  [343] = {j1=-1.508175, j2=-16.442115, j3=110.564646, j4=0.415455, j5=81.660645, j6=16.991073}
  [344] = {j1=-1.524518, j2=-16.44309, j3=110.565344, j4=0.416666, j5=81.66104, j6=16.974604}
  [345] = {j1=-1.540861, j2=-16.44406, j3=110.566039, j4=0.417877, j5=81.661434, j6=16.958135}
  [346] = {j1=-1.557205, j2=-16.445027, j3=110.566731, j4=0.419088, j5=81.661827, j6=16.941665}
  [347] = {j1=-1.573549, j2=-16.44599, j3=110.567421, j4=0.420298, j5=81.66222, j6=16.925195}
  [348] = {j1=-1.589892, j2=-16.446949, j3=110.568108, j4=0.421509, j5=81.662611, j6=16.908725}
  [349] = {j1=-1.606237, j2=-16.447904, j3=110.568792, j4=0.42272, j5=81.663002, j6=16.892255}
  [350] = {j1=-1.622581, j2=-16.448855, j3=110.569473, j4=0.423931, j5=81.663393, j6=16.875785}
  [351] = {j1=-1.638925, j2=-16.449803, j3=110.570151, j4=0.425142, j5=81.663782, j6=16.859315}
  [352] = {j1=-1.65527, j2=-16.450746, j3=110.570827, j4=0.426352, j5=81.664171, j6=16.842844}
  [353] = {j1=-1.671615, j2=-16.451685, j3=110.571499, j4=0.427563, j5=81.664559, j6=16.826373}
  [354] = {j1=-1.68796, j2=-16.452621, j3=110.572169, j4=0.428774, j5=81.664946, j6=16.809902}
  [355] = {j1=-1.704305, j2=-16.453553, j3=110.572836, j4=0.429985, j5=81.665333, j6=16.793431}
  [356] = {j1=-1.720651, j2=-16.45448, j3=110.573501, j4=0.431195, j5=81.665719, j6=16.77696}
  [357] = {j1=-1.736996, j2=-16.455404, j3=110.574162, j4=0.432406, j5=81.666104, j6=16.760488}
  [358] = {j1=-1.753342, j2=-16.456324, j3=110.574821, j4=0.433617, j5=81.666488, j6=16.744017}
  [359] = {j1=-1.769688, j2=-16.45724, j3=110.575476, j4=0.434827, j5=81.666871, j6=16.727545}
  [360] = {j1=-1.786034, j2=-16.458152, j3=110.576129, j4=0.436038, j5=81.667254, j6=16.711073}
  [361] = {j1=-1.80238, j2=-16.45906, j3=110.57678, j4=0.437248, j5=81.667636, j6=16.694601}
  [362] = {j1=-1.818727, j2=-16.459964, j3=110.577427, j4=0.438459, j5=81.668017, j6=16.678129}
  [363] = {j1=-1.835073, j2=-16.460865, j3=110.578072, j4=0.439669, j5=81.668398, j6=16.661656}
  [364] = {j1=-1.85142, j2=-16.461761, j3=110.578713, j4=0.44088, j5=81.668778, j6=16.645184}
  [365] = {j1=-1.867767, j2=-16.462654, j3=110.579352, j4=0.44209, j5=81.669157, j6=16.628711}
  [366] = {j1=-1.884114, j2=-16.463542, j3=110.579988, j4=0.443301, j5=81.669535, j6=16.612238}
  [367] = {j1=-1.900461, j2=-16.464427, j3=110.580622, j4=0.444511, j5=81.669912, j6=16.595765}
  [368] = {j1=-1.900461, j2=-16.464427, j3=110.580622, j4=0.444511, j5=81.669912, j6=16.595765}
  [369] = {j1=-1.916822, j2=-16.465308, j3=110.581253, j4=0.445722, j5=81.670289, j6=16.579279}
  [370] = {j1=-1.933183, j2=-16.466186, j3=110.581881, j4=0.446933, j5=81.670666, j6=16.562793}
  [371] = {j1=-1.949544, j2=-16.467059, j3=110.582506, j4=0.448144, j5=81.671041, j6=16.546306}
  [372] = {j1=-1.965906, j2=-16.467929, j3=110.583129, j4=0.449354, j5=81.671416, j6=16.52982}
  [373] = {j1=-1.982267, j2=-16.468795, j3=110.583748, j4=0.450565, j5=81.67179, j6=16.513333}
  [374] = {j1=-1.998629, j2=-16.469657, j3=110.584365, j4=0.451776, j5=81.672163, j6=16.496846}
  [375] = {j1=-2.014991, j2=-16.470515, j3=110.584979, j4=0.452986, j5=81.672536, j6=16.480359}
  [376] = {j1=-2.031353, j2=-16.471369, j3=110.585591, j4=0.454197, j5=81.672908, j6=16.463872}
  [377] = {j1=-2.047715, j2=-16.472219, j3=110.586199, j4=0.455408, j5=81.673279, j6=16.447385}
  [378] = {j1=-2.064077, j2=-16.473065, j3=110.586805, j4=0.456618, j5=81.673649, j6=16.430898}
  [379] = {j1=-2.080439, j2=-16.473907, j3=110.587407, j4=0.457829, j5=81.674018, j6=16.41441}
  [380] = {j1=-2.096801, j2=-16.474746, j3=110.588007, j4=0.459039, j5=81.674387, j6=16.397923}
  [381] = {j1=-2.113164, j2=-16.47558, j3=110.588604, j4=0.46025, j5=81.674755, j6=16.381435}
  [382] = {j1=-2.129526, j2=-16.47641, j3=110.589199, j4=0.46146, j5=81.675122, j6=16.364947}
  [383] = {j1=-2.145889, j2=-16.477237, j3=110.58979, j4=0.462671, j5=81.675489, j6=16.348459}
  [384] = {j1=-2.162252, j2=-16.47806, j3=110.590379, j4=0.463881, j5=81.675854, j6=16.331971}
  [385] = {j1=-2.178615, j2=-16.478878, j3=110.590965, j4=0.465092, j5=81.676219, j6=16.315483}
  [386] = {j1=-2.194978, j2=-16.479693, j3=110.591548, j4=0.466302, j5=81.676583, j6=16.298995}
  [387] = {j1=-2.211341, j2=-16.480504, j3=110.592128, j4=0.467512, j5=81.676947, j6=16.282507}
  [388] = {j1=-2.227704, j2=-16.481311, j3=110.592705, j4=0.468723, j5=81.677309, j6=16.266018}
  [389] = {j1=-2.244067, j2=-16.482114, j3=110.59328, j4=0.469933, j5=81.677671, j6=16.24953}
  [390] = {j1=-2.260431, j2=-16.482913, j3=110.593852, j4=0.471143, j5=81.678032, j6=16.233041}
  [391] = {j1=-2.276794, j2=-16.483708, j3=110.594421, j4=0.472354, j5=81.678393, j6=16.216553}
  [392] = {j1=-2.293158, j2=-16.484499, j3=110.594987, j4=0.473564, j5=81.678752, j6=16.200064}
  [393] = {j1=-2.309521, j2=-16.485286, j3=110.59555, j4=0.474774, j5=81.679111, j6=16.183575}
  [394] = {j1=-2.325885, j2=-16.48607, j3=110.596111, j4=0.475984, j5=81.679469, j6=16.167086}
  [395] = {j1=-2.342249, j2=-16.486849, j3=110.596668, j4=0.477194, j5=81.679827, j6=16.150597}
  [396] = {j1=-2.358613, j2=-16.487625, j3=110.597223, j4=0.478405, j5=81.680183, j6=16.134108}
  [397] = {j1=-2.374977, j2=-16.488396, j3=110.597775, j4=0.479615, j5=81.680539, j6=16.117619}
  [398] = {j1=-2.391341, j2=-16.489164, j3=110.598324, j4=0.480825, j5=81.680894, j6=16.10113}
  [399] = {j1=-2.407705, j2=-16.489928, j3=110.598871, j4=0.482035, j5=81.681248, j6=16.084641}
  [400] = {j1=-2.424069, j2=-16.490687, j3=110.599414, j4=0.483245, j5=81.681602, j6=16.068152}
  [401] = {j1=-2.440433, j2=-16.491443, j3=110.599955, j4=0.484455, j5=81.681955, j6=16.051662}
  [402] = {j1=-2.456798, j2=-16.492195, j3=110.600493, j4=0.485665, j5=81.682307, j6=16.035173}
  [403] = {j1=-2.473162, j2=-16.492943, j3=110.601028, j4=0.486874, j5=81.682658, j6=16.018683}
  [404] = {j1=-2.489526, j2=-16.493687, j3=110.60156, j4=0.488084, j5=81.683008, j6=16.002194}
  [405] = {j1=-2.505891, j2=-16.494427, j3=110.60209, j4=0.489294, j5=81.683358, j6=15.985704}
  [406] = {j1=-2.522255, j2=-16.495164, j3=110.602616, j4=0.490504, j5=81.683707, j6=15.969215}
  [407] = {j1=-2.53862, j2=-16.495896, j3=110.60314, j4=0.491714, j5=81.684055, j6=15.952725}
  [408] = {j1=-2.554984, j2=-16.496624, j3=110.603661, j4=0.492923, j5=81.684402, j6=15.936235}
  [409] = {j1=-2.571349, j2=-16.497349, j3=110.604179, j4=0.494133, j5=81.684749, j6=15.919746}
  [410] = {j1=-2.587713, j2=-16.498069, j3=110.604695, j4=0.495343, j5=81.685095, j6=15.903256}
  [411] = {j1=-2.604078, j2=-16.498786, j3=110.605207, j4=0.496552, j5=81.68544, j6=15.886766}
  [412] = {j1=-2.620443, j2=-16.499498, j3=110.605717, j4=0.497762, j5=81.685784, j6=15.870276}
  [413] = {j1=-2.636808, j2=-16.500207, j3=110.606224, j4=0.498972, j5=81.686128, j6=15.853787}
  [414] = {j1=-2.653172, j2=-16.500912, j3=110.606728, j4=0.500181, j5=81.68647, j6=15.837297}
  [415] = {j1=-2.669537, j2=-16.501613, j3=110.607229, j4=0.501391, j5=81.686812, j6=15.820807}
  [416] = {j1=-2.685902, j2=-16.502309, j3=110.607728, j4=0.5026, j5=81.687154, j6=15.804317}
  [417] = {j1=-2.702267, j2=-16.503002, j3=110.608223, j4=0.503809, j5=81.687494, j6=15.787827}
  [418] = {j1=-2.718632, j2=-16.503691, j3=110.608716, j4=0.505019, j5=81.687834, j6=15.771337}
  [419] = {j1=-2.734996, j2=-16.504377, j3=110.609206, j4=0.506228, j5=81.688173, j6=15.754847}
  [420] = {j1=-2.751361, j2=-16.505058, j3=110.609693, j4=0.507437, j5=81.688511, j6=15.738357}
  [421] = {j1=-2.767726, j2=-16.505735, j3=110.610177, j4=0.508647, j5=81.688848, j6=15.721867}
  [422] = {j1=-2.784091, j2=-16.506408, j3=110.610659, j4=0.509856, j5=81.689185, j6=15.705377}
  [423] = {j1=-2.800456, j2=-16.507078, j3=110.611138, j4=0.511065, j5=81.689521, j6=15.688887}
  [424] = {j1=-2.816821, j2=-16.507743, j3=110.611613, j4=0.512274, j5=81.689856, j6=15.672397}
  [425] = {j1=-2.833186, j2=-16.508405, j3=110.612086, j4=0.513483, j5=81.69019, j6=15.655908}
  [426] = {j1=-2.84955, j2=-16.509062, j3=110.612557, j4=0.514693, j5=81.690524, j6=15.639418}
  [427] = {j1=-2.865915, j2=-16.509716, j3=110.613024, j4=0.515902, j5=81.690857, j6=15.622928}
  [428] = {j1=-2.88228, j2=-16.510365, j3=110.613489, j4=0.517111, j5=81.691189, j6=15.606438}
  [429] = {j1=-2.898645, j2=-16.511011, j3=110.61395, j4=0.51832, j5=81.69152, j6=15.589948}
  [430] = {j1=-2.91501, j2=-16.511653, j3=110.614409, j4=0.519528, j5=81.691851, j6=15.573458}
  [431] = {j1=-2.931375, j2=-16.512291, j3=110.614865, j4=0.520737, j5=81.69218, j6=15.556968}
  [432] = {j1=-2.947739, j2=-16.512925, j3=110.615319, j4=0.521946, j5=81.692509, j6=15.540478}
  [433] = {j1=-2.964104, j2=-16.513555, j3=110.615769, j4=0.523155, j5=81.692837, j6=15.523989}
  [434] = {j1=-2.980469, j2=-16.514181, j3=110.616217, j4=0.524364, j5=81.693165, j6=15.507499}
  [435] = {j1=-2.996834, j2=-16.514803, j3=110.616662, j4=0.525573, j5=81.693491, j6=15.491009}
  [436] = {j1=-3.013198, j2=-16.515421, j3=110.617104, j4=0.526781, j5=81.693817, j6=15.474519}
  [437] = {j1=-3.029563, j2=-16.516035, j3=110.617543, j4=0.52799, j5=81.694142, j6=15.45803}
  [438] = {j1=-3.045927, j2=-16.516646, j3=110.617979, j4=0.529198, j5=81.694467, j6=15.44154}
  [439] = {j1=-3.062292, j2=-16.517252, j3=110.618413, j4=0.530407, j5=81.69479, j6=15.42505}
  [440] = {j1=-3.078656, j2=-16.517855, j3=110.618844, j4=0.531616, j5=81.695113, j6=15.408561}
  [441] = {j1=-3.095021, j2=-16.518453, j3=110.619271, j4=0.532824, j5=81.695435, j6=15.392071}
  [442] = {j1=-3.111385, j2=-16.519048, j3=110.619697, j4=0.534032, j5=81.695756, j6=15.375582}
  [443] = {j1=-3.12775, j2=-16.519638, j3=110.620119, j4=0.535241, j5=81.696077, j6=15.359093}
  [444] = {j1=-3.144114, j2=-16.520225, j3=110.620538, j4=0.536449, j5=81.696396, j6=15.342603}
  [445] = {j1=-3.160478, j2=-16.520808, j3=110.620955, j4=0.537657, j5=81.696715, j6=15.326114}
  [446] = {j1=-3.176842, j2=-16.521387, j3=110.621369, j4=0.538866, j5=81.697033, j6=15.309625}
  [447] = {j1=-3.193207, j2=-16.521962, j3=110.62178, j4=0.540074, j5=81.697351, j6=15.293136}
  [448] = {j1=-3.209571, j2=-16.522532, j3=110.622188, j4=0.541282, j5=81.697667, j6=15.276647}
  [449] = {j1=-3.225935, j2=-16.523099, j3=110.622593, j4=0.54249, j5=81.697983, j6=15.260158}
  [450] = {j1=-3.242299, j2=-16.523663, j3=110.622996, j4=0.543698, j5=81.698298, j6=15.243669}
  [451] = {j1=-3.258662, j2=-16.524222, j3=110.623395, j4=0.544906, j5=81.698612, j6=15.22718}
  [452] = {j1=-3.275026, j2=-16.524777, j3=110.623792, j4=0.546114, j5=81.698926, j6=15.210691}
  [453] = {j1=-3.29139, j2=-16.525328, j3=110.624186, j4=0.547322, j5=81.699239, j6=15.194202}
  [454] = {j1=-3.307753, j2=-16.525875, j3=110.624577, j4=0.54853, j5=81.69955, j6=15.177714}
  [455] = {j1=-3.324117, j2=-16.526419, j3=110.624966, j4=0.549738, j5=81.699862, j6=15.161225}
  [456] = {j1=-3.34048, j2=-16.526958, j3=110.625351, j4=0.550946, j5=81.700172, j6=15.144737}
  [457] = {j1=-3.356844, j2=-16.527494, j3=110.625734, j4=0.552154, j5=81.700482, j6=15.128248}
  [458] = {j1=-3.373207, j2=-16.528025, j3=110.626114, j4=0.553361, j5=81.70079, j6=15.11176}
  [459] = {j1=-3.38957, j2=-16.528553, j3=110.626491, j4=0.554569, j5=81.701098, j6=15.095272}
  [460] = {j1=-3.405933, j2=-16.529077, j3=110.626866, j4=0.555776, j5=81.701406, j6=15.078784}
  [461] = {j1=-3.422296, j2=-16.529596, j3=110.627237, j4=0.556984, j5=81.701712, j6=15.062296}
  [462] = {j1=-3.438659, j2=-16.530112, j3=110.627606, j4=0.558192, j5=81.702018, j6=15.045808}
  [463] = {j1=-3.455022, j2=-16.530624, j3=110.627972, j4=0.559399, j5=81.702323, j6=15.02932}
  [464] = {j1=-3.471385, j2=-16.531132, j3=110.628335, j4=0.560606, j5=81.702627, j6=15.012832}
  [465] = {j1=-3.487747, j2=-16.531636, j3=110.628695, j4=0.561814, j5=81.70293, j6=14.996345}
  [466] = {j1=-3.50411, j2=-16.532136, j3=110.629052, j4=0.563021, j5=81.703233, j6=14.979857}
  [467] = {j1=-3.520472, j2=-16.532632, j3=110.629407, j4=0.564228, j5=81.703535, j6=14.96337}
  [468] = {j1=-3.536834, j2=-16.533124, j3=110.629758, j4=0.565436, j5=81.703836, j6=14.946883}
  [469] = {j1=-3.553196, j2=-16.533612, j3=110.630107, j4=0.566643, j5=81.704136, j6=14.930396}
  [470] = {j1=-3.569558, j2=-16.534096, j3=110.630453, j4=0.56785, j5=81.704436, j6=14.913909}
  [471] = {j1=-3.58592, j2=-16.534577, j3=110.630797, j4=0.569057, j5=81.704734, j6=14.897422}
  [472] = {j1=-3.602282, j2=-16.535053, j3=110.631137, j4=0.570264, j5=81.705032, j6=14.880935}
  [473] = {j1=-3.618643, j2=-16.535526, j3=110.631475, j4=0.571471, j5=81.70533, j6=14.864449}
  [474] = {j1=-3.635005, j2=-16.535994, j3=110.63181, j4=0.572678, j5=81.705626, j6=14.847962}
  [475] = {j1=-3.651366, j2=-16.536459, j3=110.632141, j4=0.573885, j5=81.705922, j6=14.831476}
  [476] = {j1=-3.667727, j2=-16.536919, j3=110.632471, j4=0.575091, j5=81.706216, j6=14.81499}
  [477] = {j1=-3.684088, j2=-16.537376, j3=110.632797, j4=0.576298, j5=81.70651, j6=14.798504}
  [478] = {j1=-3.700449, j2=-16.537829, j3=110.63312, j4=0.577505, j5=81.706804, j6=14.782018}
  [479] = {j1=-3.71681, j2=-16.538277, j3=110.633441, j4=0.578711, j5=81.707096, j6=14.765532}
  [480] = {j1=-3.733171, j2=-16.538722, j3=110.633759, j4=0.579918, j5=81.707388, j6=14.749047}
  [481] = {j1=-3.749531, j2=-16.539163, j3=110.634074, j4=0.581125, j5=81.707679, j6=14.732561}
  [482] = {j1=-3.765891, j2=-16.5396, j3=110.634386, j4=0.582331, j5=81.707969, j6=14.716076}
  [483] = {j1=-3.782251, j2=-16.540033, j3=110.634696, j4=0.583537, j5=81.708258, j6=14.699591}
  [484] = {j1=-3.798611, j2=-16.540462, j3=110.635002, j4=0.584744, j5=81.708547, j6=14.683106}
  [485] = {j1=-3.814971, j2=-16.540887, j3=110.635306, j4=0.58595, j5=81.708835, j6=14.666621}
  [486] = {j1=-3.831331, j2=-16.541308, j3=110.635607, j4=0.587156, j5=81.709122, j6=14.650137}
  [487] = {j1=-3.84769, j2=-16.541725, j3=110.635905, j4=0.588363, j5=81.709408, j6=14.633652}
  [488] = {j1=-3.86405, j2=-16.542139, j3=110.6362, j4=0.589569, j5=81.709693, j6=14.617168}
  [489] = {j1=-3.880409, j2=-16.542548, j3=110.636493, j4=0.590775, j5=81.709978, j6=14.600684}
  [490] = {j1=-3.896768, j2=-16.542953, j3=110.636783, j4=0.591981, j5=81.710262, j6=14.5842}
  [491] = {j1=-3.913126, j2=-16.543355, j3=110.637069, j4=0.593187, j5=81.710545, j6=14.567716}
  [492] = {j1=-3.929485, j2=-16.543752, j3=110.637353, j4=0.594393, j5=81.710827, j6=14.551233}
  [493] = {j1=-3.945843, j2=-16.544146, j3=110.637635, j4=0.595599, j5=81.711109, j6=14.534749}
  [494] = {j1=-3.962202, j2=-16.544536, j3=110.637913, j4=0.596804, j5=81.71139, j6=14.518266}
  [495] = {j1=-3.97856, j2=-16.544921, j3=110.638189, j4=0.59801, j5=81.71167, j6=14.501783}
  [496] = {j1=-3.994917, j2=-16.545303, j3=110.638461, j4=0.599216, j5=81.711949, j6=14.4853}
  [497] = {j1=-4.011275, j2=-16.545681, j3=110.638731, j4=0.600421, j5=81.712227, j6=14.468818}
  [498] = {j1=-4.027633, j2=-16.546054, j3=110.638998, j4=0.601627, j5=81.712505, j6=14.452335}
  [499] = {j1=-4.04399, j2=-16.546424, j3=110.639262, j4=0.602832, j5=81.712782, j6=14.435853}
  [500] = {j1=-4.060347, j2=-16.54679, j3=110.639524, j4=0.604038, j5=81.713058, j6=14.419371}
  [501] = {j1=-4.076704, j2=-16.547152, j3=110.639783, j4=0.605243, j5=81.713333, j6=14.402889}
  [502] = {j1=-4.09306, j2=-16.54751, j3=110.640038, j4=0.606449, j5=81.713608, j6=14.386408}
  [503] = {j1=-4.109417, j2=-16.547864, j3=110.640291, j4=0.607654, j5=81.713881, j6=14.369926}
  [504] = {j1=-4.125773, j2=-16.548214, j3=110.640541, j4=0.608859, j5=81.714154, j6=14.353445}
  [505] = {j1=-4.142129, j2=-16.548561, j3=110.640789, j4=0.610064, j5=81.714426, j6=14.336964}
  [506] = {j1=-4.158485, j2=-16.548903, j3=110.641033, j4=0.611269, j5=81.714698, j6=14.320483}
  [507] = {j1=-4.17484, j2=-16.549241, j3=110.641275, j4=0.612474, j5=81.714968, j6=14.304003}
  [508] = {j1=-4.191195, j2=-16.549576, j3=110.641514, j4=0.613679, j5=81.715238, j6=14.287523}
  [509] = {j1=-4.20755, j2=-16.549906, j3=110.64175, j4=0.614884, j5=81.715507, j6=14.271043}
  [510] = {j1=-4.223905, j2=-16.550232, j3=110.641983, j4=0.616089, j5=81.715775, j6=14.254563}
  [511] = {j1=-4.24026, j2=-16.550555, j3=110.642214, j4=0.617294, j5=81.716043, j6=14.238083}
  [512] = {j1=-4.256614, j2=-16.550873, j3=110.642441, j4=0.618498, j5=81.716309, j6=14.221604}
  [513] = {j1=-4.272968, j2=-16.551188, j3=110.642666, j4=0.619703, j5=81.716575, j6=14.205125}
  [514] = {j1=-4.289322, j2=-16.551499, j3=110.642888, j4=0.620908, j5=81.71684, j6=14.188646}
  [515] = {j1=-4.305676, j2=-16.551805, j3=110.643107, j4=0.622112, j5=81.717105, j6=14.172167}
  [516] = {j1=-4.322029, j2=-16.552108, j3=110.643323, j4=0.623317, j5=81.717368, j6=14.155689}
  [517] = {j1=-4.338383, j2=-16.552407, j3=110.643537, j4=0.624521, j5=81.717631, j6=14.139211}
  [518] = {j1=-4.354736, j2=-16.552702, j3=110.643747, j4=0.625725, j5=81.717893, j6=14.122733}
  [519] = {j1=-4.371088, j2=-16.552993, j3=110.643955, j4=0.62693, j5=81.718154, j6=14.106255}
  [520] = {j1=-4.387441, j2=-16.55328, j3=110.64416, j4=0.628134, j5=81.718414, j6=14.089778}
  [521] = {j1=-4.403793, j2=-16.553563, j3=110.644362, j4=0.629338, j5=81.718674, j6=14.073301}
  [522] = {j1=-4.420145, j2=-16.553842, j3=110.644562, j4=0.630542, j5=81.718933, j6=14.056824}
  [523] = {j1=-4.436496, j2=-16.554117, j3=110.644758, j4=0.631746, j5=81.719191, j6=14.040347}
  [524] = {j1=-4.452848, j2=-16.554388, j3=110.644952, j4=0.63295, j5=81.719448, j6=14.023871}
  [525] = {j1=-4.469199, j2=-16.554655, j3=110.645143, j4=0.634154, j5=81.719704, j6=14.007395}
  [526] = {j1=-4.485549, j2=-16.554919, j3=110.645331, j4=0.635357, j5=81.71996, j6=13.990919}
  [527] = {j1=-4.5019, j2=-16.555178, j3=110.645516, j4=0.636561, j5=81.720215, j6=13.974444}
  [528] = {j1=-4.51825, j2=-16.555433, j3=110.645699, j4=0.637765, j5=81.720469, j6=13.957968}
  [529] = {j1=-4.5346, j2=-16.555685, j3=110.645878, j4=0.638968, j5=81.720722, j6=13.941493}
  [530] = {j1=-4.55095, j2=-16.555932, j3=110.646055, j4=0.640172, j5=81.720975, j6=13.925019}
  [531] = {j1=-4.567299, j2=-16.556176, j3=110.646229, j4=0.641375, j5=81.721226, j6=13.908544}
  [532] = {j1=-4.583648, j2=-16.556416, j3=110.6464, j4=0.642579, j5=81.721477, j6=13.89207}
  [533] = {j1=-4.599997, j2=-16.556651, j3=110.646568, j4=0.643782, j5=81.721727, j6=13.875596}
  [534] = {j1=-4.616346, j2=-16.556883, j3=110.646734, j4=0.644985, j5=81.721977, j6=13.859123}
  [535] = {j1=-4.632694, j2=-16.557111, j3=110.646896, j4=0.646189, j5=81.722225, j6=13.84265}
  [536] = {j1=-4.649042, j2=-16.557334, j3=110.647056, j4=0.647392, j5=81.722473, j6=13.826177}
  [537] = {j1=-4.66539, j2=-16.557554, j3=110.647213, j4=0.648595, j5=81.72272, j6=13.809704}
  [538] = {j1=-4.681737, j2=-16.55777, j3=110.647368, j4=0.649798, j5=81.722966, j6=13.793232}
  [539] = {j1=-4.698084, j2=-16.557982, j3=110.647519, j4=0.651, j5=81.723212, j6=13.77676}
  [540] = {j1=-4.714431, j2=-16.55819, j3=110.647668, j4=0.652203, j5=81.723456, j6=13.760288}
  [541] = {j1=-4.730777, j2=-16.558394, j3=110.647813, j4=0.653406, j5=81.7237, j6=13.743817}
  [542] = {j1=-4.747123, j2=-16.558594, j3=110.647956, j4=0.654609, j5=81.723943, j6=13.727346}
  [543] = {j1=-4.763469, j2=-16.55879, j3=110.648096, j4=0.655811, j5=81.724185, j6=13.710875}
  [544] = {j1=-4.779814, j2=-16.558983, j3=110.648234, j4=0.657014, j5=81.724427, j6=13.694405}
  [545] = {j1=-4.796159, j2=-16.559171, j3=110.648368, j4=0.658216, j5=81.724667, j6=13.677934}
  [546] = {j1=-4.812504, j2=-16.559355, j3=110.6485, j4=0.659419, j5=81.724907, j6=13.661465}
  [547] = {j1=-4.828849, j2=-16.559535, j3=110.648628, j4=0.660621, j5=81.725146, j6=13.644995}
  [548] = {j1=-4.845193, j2=-16.559712, j3=110.648754, j4=0.661823, j5=81.725385, j6=13.628526}
  [549] = {j1=-4.861536, j2=-16.559884, j3=110.648878, j4=0.663025, j5=81.725622, j6=13.612057}
  [550] = {j1=-4.87788, j2=-16.560053, j3=110.648998, j4=0.664228, j5=81.725859, j6=13.595589}
  [551] = {j1=-4.894223, j2=-16.560217, j3=110.649115, j4=0.66543, j5=81.726095, j6=13.579121}
  [552] = {j1=-4.910566, j2=-16.560378, j3=110.64923, j4=0.666632, j5=81.72633, j6=13.562653}
  [553] = {j1=-4.926908, j2=-16.560535, j3=110.649342, j4=0.667833, j5=81.726564, j6=13.546185}
  [554] = {j1=-4.94325, j2=-16.560687, j3=110.649451, j4=0.669035, j5=81.726798, j6=13.529718}
  [555] = {j1=-4.959592, j2=-16.560836, j3=110.649557, j4=0.670237, j5=81.727031, j6=13.513252}
  [556] = {j1=-4.975933, j2=-16.560981, j3=110.649661, j4=0.671439, j5=81.727262, j6=13.496785}
  [557] = {j1=-4.992274, j2=-16.561122, j3=110.649761, j4=0.67264, j5=81.727494, j6=13.480319}
  [558] = {j1=-5.008615, j2=-16.561258, j3=110.649859, j4=0.673842, j5=81.727724, j6=13.463853}
  [559] = {j1=-5.024955, j2=-16.561391, j3=110.649954, j4=0.675043, j5=81.727954, j6=13.447388}
  [560] = {j1=-5.041295, j2=-16.56152, j3=110.650046, j4=0.676244, j5=81.728182, j6=13.430923}
  [561] = {j1=-5.057635, j2=-16.561645, j3=110.650135, j4=0.677446, j5=81.72841, j6=13.414459}
  [562] = {j1=-5.073974, j2=-16.561766, j3=110.650222, j4=0.678647, j5=81.728638, j6=13.397994}
  [563] = {j1=-5.090313, j2=-16.561884, j3=110.650306, j4=0.679848, j5=81.728864, j6=13.381531}
  [564] = {j1=-5.106651, j2=-16.561997, j3=110.650386, j4=0.681049, j5=81.72909, j6=13.365067}
  [565] = {j1=-5.12299, j2=-16.562106, j3=110.650464, j4=0.68225, j5=81.729315, j6=13.348604}
  [566] = {j1=-5.139327, j2=-16.562211, j3=110.65054, j4=0.683451, j5=81.729539, j6=13.332141}
  [567] = {j1=-5.155665, j2=-16.562313, j3=110.650612, j4=0.684652, j5=81.729762, j6=13.315679}
  [568] = {j1=-5.172002, j2=-16.56241, j3=110.650681, j4=0.685852, j5=81.729984, j6=13.299217}
  [569] = {j1=-5.188338, j2=-16.562503, j3=110.650748, j4=0.687053, j5=81.730206, j6=13.282755}
  [570] = {j1=-5.204674, j2=-16.562593, j3=110.650812, j4=0.688253, j5=81.730427, j6=13.266294}
  [571] = {j1=-5.22101, j2=-16.562678, j3=110.650873, j4=0.689454, j5=81.730647, j6=13.249833}
  [572] = {j1=-5.237345, j2=-16.56276, j3=110.650931, j4=0.690654, j5=81.730866, j6=13.233373}
  [573] = {j1=-5.25368, j2=-16.562838, j3=110.650987, j4=0.691855, j5=81.731085, j6=13.216913}
  [574] = {j1=-5.270015, j2=-16.562911, j3=110.651039, j4=0.693055, j5=81.731303, j6=13.200453}
  [575] = {j1=-5.286349, j2=-16.562981, j3=110.651089, j4=0.694255, j5=81.731519, j6=13.183994}
  [576] = {j1=-5.302683, j2=-16.563047, j3=110.651136, j4=0.695455, j5=81.731736, j6=13.167535}
  [577] = {j1=-5.319016, j2=-16.563109, j3=110.65118, j4=0.696655, j5=81.731951, j6=13.151077}
  [578] = {j1=-5.335349, j2=-16.563166, j3=110.651222, j4=0.697855, j5=81.732165, j6=13.134619}
  [579] = {j1=-5.351682, j2=-16.56322, j3=110.65126, j4=0.699055, j5=81.732379, j6=13.118161}
  [580] = {j1=-5.368014, j2=-16.56327, j3=110.651296, j4=0.700255, j5=81.732592, j6=13.101704}
  [581] = {j1=-5.384346, j2=-16.563316, j3=110.651329, j4=0.701454, j5=81.732804, j6=13.085247}
  [582] = {j1=-5.400677, j2=-16.563358, j3=110.651359, j4=0.702654, j5=81.733016, j6=13.068791}
  [583] = {j1=-5.417008, j2=-16.563397, j3=110.651386, j4=0.703853, j5=81.733226, j6=13.052335}
  [584] = {j1=-5.433338, j2=-16.563431, j3=110.65141, j4=0.705053, j5=81.733436, j6=13.035879}
  [585] = {j1=-5.449668, j2=-16.563461, j3=110.651432, j4=0.706252, j5=81.733645, j6=13.019424}
  [586] = {j1=-5.465998, j2=-16.563487, j3=110.651451, j4=0.707451, j5=81.733853, j6=13.00297}
  [587] = {j1=-5.482327, j2=-16.563509, j3=110.651467, j4=0.70865, j5=81.734061, j6=12.986516}
  [588] = {j1=-5.498655, j2=-16.563528, j3=110.65148, j4=0.70985, j5=81.734267, j6=12.970062}
  [589] = {j1=-5.514984, j2=-16.563542, j3=110.65149, j4=0.711049, j5=81.734473, j6=12.953608}
  [590] = {j1=-5.531311, j2=-16.563553, j3=110.651497, j4=0.712247, j5=81.734678, j6=12.937156}
  [591] = {j1=-5.547639, j2=-16.563559, j3=110.651502, j4=0.713446, j5=81.734882, j6=12.920703}
  [592] = {j1=-5.563966, j2=-16.563562, j3=110.651504, j4=0.714645, j5=81.735086, j6=12.904251}
  [593] = {j1=-5.580292, j2=-16.56356, j3=110.651503, j4=0.715844, j5=81.735288, j6=12.8878}
  [594] = {j1=-5.596618, j2=-16.563555, j3=110.651499, j4=0.717042, j5=81.73549, j6=12.871348}
  [595] = {j1=-5.612944, j2=-16.563546, j3=110.651492, j4=0.718241, j5=81.735691, j6=12.854898}
  [596] = {j1=-5.629269, j2=-16.563532, j3=110.651483, j4=0.719439, j5=81.735892, j6=12.838448}
  [597] = {j1=-5.645593, j2=-16.563515, j3=110.651471, j4=0.720637, j5=81.736091, j6=12.821998}
  [598] = {j1=-5.661918, j2=-16.563494, j3=110.651455, j4=0.721836, j5=81.73629, j6=12.805549}
  [599] = {j1=-5.678241, j2=-16.563469, j3=110.651437, j4=0.723034, j5=81.736487, j6=12.7891}
  [600] = {j1=-5.694565, j2=-16.56344, j3=110.651417, j4=0.724232, j5=81.736685, j6=12.772651}
  [601] = {j1=-5.710887, j2=-16.563407, j3=110.651393, j4=0.72543, j5=81.736881, j6=12.756204}
  [602] = {j1=-5.72721, j2=-16.56337, j3=110.651367, j4=0.726628, j5=81.737076, j6=12.739756}
  [603] = {j1=-5.743531, j2=-16.563329, j3=110.651337, j4=0.727825, j5=81.737271, j6=12.723309}
  [604] = {j1=-5.759853, j2=-16.563284, j3=110.651305, j4=0.729023, j5=81.737465, j6=12.706863}
  [605] = {j1=-5.776174, j2=-16.563235, j3=110.651271, j4=0.730221, j5=81.737658, j6=12.690417}
  [606] = {j1=-5.792494, j2=-16.563182, j3=110.651233, j4=0.731418, j5=81.73785, j6=12.673971}
  [607] = {j1=-5.808814, j2=-16.563126, j3=110.651192, j4=0.732616, j5=81.738042, j6=12.657526}
  [608] = {j1=-5.825133, j2=-16.563065, j3=110.651149, j4=0.733813, j5=81.738233, j6=12.641082}
  [609] = {j1=-5.841452, j2=-16.563, j3=110.651103, j4=0.73501, j5=81.738422, j6=12.624638}
  [610] = {j1=-5.85777, j2=-16.562932, j3=110.651054, j4=0.736207, j5=81.738612, j6=12.608194}
  [611] = {j1=-5.874088, j2=-16.562859, j3=110.651002, j4=0.737404, j5=81.7388, j6=12.591751}
  [612] = {j1=-5.890406, j2=-16.562783, j3=110.650947, j4=0.738601, j5=81.738987, j6=12.575309}
  [613] = {j1=-5.906723, j2=-16.562702, j3=110.65089, j4=0.739798, j5=81.739174, j6=12.558867}
  [614] = {j1=-5.923039, j2=-16.562618, j3=110.65083, j4=0.740995, j5=81.73936, j6=12.542425}
  [615] = {j1=-5.939355, j2=-16.562529, j3=110.650767, j4=0.742192, j5=81.739545, j6=12.525984}
  [616] = {j1=-5.95567, j2=-16.562437, j3=110.650701, j4=0.743388, j5=81.73973, j6=12.509544}
  [617] = {j1=-5.971985, j2=-16.562341, j3=110.650632, j4=0.744585, j5=81.739913, j6=12.493104}
  [618] = {j1=-5.988299, j2=-16.562241, j3=110.65056, j4=0.745781, j5=81.740096, j6=12.476664}
  [619] = {j1=-6.004613, j2=-16.562137, j3=110.650486, j4=0.746977, j5=81.740278, j6=12.460225}
  [620] = {j1=-6.020926, j2=-16.562029, j3=110.650409, j4=0.748174, j5=81.740459, j6=12.443787}
  [621] = {j1=-6.037239, j2=-16.561916, j3=110.650329, j4=0.74937, j5=81.740639, j6=12.427349}
  [622] = {j1=-6.053551, j2=-16.5618, j3=110.650246, j4=0.750566, j5=81.740819, j6=12.410911}
  [623] = {j1=-6.069863, j2=-16.561681, j3=110.65016, j4=0.751762, j5=81.740998, j6=12.394474}
  [624] = {j1=-6.086174, j2=-16.561557, j3=110.650072, j4=0.752958, j5=81.741176, j6=12.378038}
  [625] = {j1=-6.102485, j2=-16.561429, j3=110.64998, j4=0.754153, j5=81.741353, j6=12.361602}
  [626] = {j1=-6.118795, j2=-16.561297, j3=110.649886, j4=0.755349, j5=81.741529, j6=12.345167}
  [627] = {j1=-6.135104, j2=-16.561161, j3=110.649789, j4=0.756545, j5=81.741705, j6=12.328732}
  [628] = {j1=-6.151413, j2=-16.561021, j3=110.649689, j4=0.75774, j5=81.74188, j6=12.312298}
  [629] = {j1=-6.167722, j2=-16.560878, j3=110.649587, j4=0.758935, j5=81.742054, j6=12.295864}
  [630] = {j1=-6.18403, j2=-16.56073, j3=110.649481, j4=0.760131, j5=81.742227, j6=12.279431}
  [631] = {j1=-6.200337, j2=-16.560579, j3=110.649373, j4=0.761326, j5=81.742399, j6=12.262999}
  [632] = {j1=-6.216644, j2=-16.560423, j3=110.649262, j4=0.762521, j5=81.742571, j6=12.246567}
  [633] = {j1=-6.23295, j2=-16.560264, j3=110.649148, j4=0.763716, j5=81.742742, j6=12.230135}
  [634] = {j1=-6.249256, j2=-16.5601, j3=110.649031, j4=0.764911, j5=81.742912, j6=12.213704}
  [635] = {j1=-6.265561, j2=-16.559933, j3=110.648912, j4=0.766106, j5=81.743081, j6=12.197274}
  [636] = {j1=-6.281866, j2=-16.559762, j3=110.64879, j4=0.7673, j5=81.74325, j6=12.180844}
  [637] = {j1=-6.29817, j2=-16.559586, j3=110.648664, j4=0.768495, j5=81.743417, j6=12.164415}
  [638] = {j1=-6.314473, j2=-16.559407, j3=110.648536, j4=0.769689, j5=81.743584, j6=12.147986}
  [639] = {j1=-6.330776, j2=-16.559224, j3=110.648405, j4=0.770884, j5=81.74375, j6=12.131558}
  [640] = {j1=-6.347078, j2=-16.559037, j3=110.648272, j4=0.772078, j5=81.743915, j6=12.115131}
  [641] = {j1=-6.36338, j2=-16.558846, j3=110.648135, j4=0.773272, j5=81.74408, j6=12.098704}
  [642] = {j1=-6.379681, j2=-16.558651, j3=110.647996, j4=0.774466, j5=81.744243, j6=12.082277}
  [643] = {j1=-6.395981, j2=-16.558452, j3=110.647854, j4=0.77566, j5=81.744406, j6=12.065851}
  [644] = {j1=-6.412281, j2=-16.558249, j3=110.647709, j4=0.776854, j5=81.744568, j6=12.049426}
  [645] = {j1=-6.428581, j2=-16.558042, j3=110.647561, j4=0.778048, j5=81.74473, j6=12.033002}
  [646] = {j1=-6.444879, j2=-16.557831, j3=110.647411, j4=0.779242, j5=81.74489, j6=12.016578}
  [647] = {j1=-6.461178, j2=-16.557616, j3=110.647257, j4=0.780435, j5=81.74505, j6=12.000154}
  [648] = {j1=-6.477475, j2=-16.557398, j3=110.647101, j4=0.781629, j5=81.745209, j6=11.983731}
  [649] = {j1=-6.493772, j2=-16.557175, j3=110.646942, j4=0.782822, j5=81.745367, j6=11.967309}
  [650] = {j1=-6.510069, j2=-16.556948, j3=110.64678, j4=0.784015, j5=81.745524, j6=11.950887}
  [651] = {j1=-6.526364, j2=-16.556718, j3=110.646615, j4=0.785209, j5=81.74568, j6=11.934466}
  [652] = {j1=-6.542659, j2=-16.556483, j3=110.646448, j4=0.786402, j5=81.745836, j6=11.918046}
  [653] = {j1=-6.558954, j2=-16.556245, j3=110.646277, j4=0.787595, j5=81.745991, j6=11.901626}
  [654] = {j1=-6.575248, j2=-16.556003, j3=110.646104, j4=0.788787, j5=81.746145, j6=11.885207}
  [655] = {j1=-6.591541, j2=-16.555756, j3=110.645928, j4=0.78998, j5=81.746298, j6=11.868788}
  [656] = {j1=-6.607834, j2=-16.555506, j3=110.64575, j4=0.791173, j5=81.746451, j6=11.85237}
  [657] = {j1=-6.624126, j2=-16.555252, j3=110.645568, j4=0.792365, j5=81.746603, j6=11.835952}
  [658] = {j1=-6.640418, j2=-16.554993, j3=110.645383, j4=0.793558, j5=81.746753, j6=11.819536}
  [659] = {j1=-6.656708, j2=-16.554731, j3=110.645196, j4=0.79475, j5=81.746904, j6=11.803119}
  [660] = {j1=-6.672999, j2=-16.554465, j3=110.645006, j4=0.795943, j5=81.747053, j6=11.786704}
  [661] = {j1=-6.689288, j2=-16.554195, j3=110.644813, j4=0.797135, j5=81.747201, j6=11.770289}
  [662] = {j1=-6.705577, j2=-16.553921, j3=110.644617, j4=0.798327, j5=81.747349, j6=11.753875}
  [663] = {j1=-6.721865, j2=-16.553643, j3=110.644419, j4=0.799519, j5=81.747496, j6=11.737461}
  [664] = {j1=-6.738153, j2=-16.553361, j3=110.644217, j4=0.80071, j5=81.747642, j6=11.721048}
  [665] = {j1=-6.75444, j2=-16.553075, j3=110.644013, j4=0.801902, j5=81.747787, j6=11.704636}
  [666] = {j1=-6.770727, j2=-16.552786, j3=110.643806, j4=0.803094, j5=81.747932, j6=11.688224}
  [667] = {j1=-6.787012, j2=-16.552492, j3=110.643596, j4=0.804285, j5=81.748076, j6=11.671813}
  [668] = {j1=-6.803297, j2=-16.552194, j3=110.643384, j4=0.805477, j5=81.748219, j6=11.655402}
  [669] = {j1=-6.819582, j2=-16.551892, j3=110.643168, j4=0.806668, j5=81.748361, j6=11.638992}
  [670] = {j1=-6.835866, j2=-16.551587, j3=110.64295, j4=0.807859, j5=81.748502, j6=11.622583}
  [671] = {j1=-6.852149, j2=-16.551277, j3=110.642729, j4=0.80905, j5=81.748643, j6=11.606175}
  [672] = {j1=-6.868431, j2=-16.550964, j3=110.642505, j4=0.810241, j5=81.748782, j6=11.589767}
  [673] = {j1=-6.884713, j2=-16.550646, j3=110.642278, j4=0.811432, j5=81.748921, j6=11.573359}
  [674] = {j1=-6.900994, j2=-16.550325, j3=110.642048, j4=0.812623, j5=81.749059, j6=11.556953}
  [675] = {j1=-6.917275, j2=-16.55, j3=110.641816, j4=0.813814, j5=81.749197, j6=11.540547}
  [676] = {j1=-6.933554, j2=-16.54967, j3=110.641581, j4=0.815004, j5=81.749333, j6=11.524142}
  [677] = {j1=-6.949834, j2=-16.549337, j3=110.641343, j4=0.816195, j5=81.749469, j6=11.507737}
  [678] = {j1=-6.966112, j2=-16.549, j3=110.641102, j4=0.817385, j5=81.749604, j6=11.491333}
  [679] = {j1=-6.98239, j2=-16.548659, j3=110.640858, j4=0.818575, j5=81.749738, j6=11.47493}
  [680] = {j1=-6.998667, j2=-16.548314, j3=110.640612, j4=0.819765, j5=81.749872, j6=11.458528}
  [681] = {j1=-7.014943, j2=-16.547965, j3=110.640362, j4=0.820955, j5=81.750004, j6=11.442126}
  [682] = {j1=-7.031219, j2=-16.547612, j3=110.64011, j4=0.822145, j5=81.750136, j6=11.425724}
  [683] = {j1=-7.047494, j2=-16.547255, j3=110.639855, j4=0.823335, j5=81.750267, j6=11.409324}
  [684] = {j1=-7.063769, j2=-16.546894, j3=110.639597, j4=0.824524, j5=81.750397, j6=11.392924}
  [685] = {j1=-7.080042, j2=-16.546529, j3=110.639336, j4=0.825714, j5=81.750526, j6=11.376525}
  [686] = {j1=-7.096315, j2=-16.546161, j3=110.639073, j4=0.826903, j5=81.750655, j6=11.360126}
  [687] = {j1=-7.112587, j2=-16.545788, j3=110.638807, j4=0.828093, j5=81.750783, j6=11.343729}
  [688] = {j1=-7.128859, j2=-16.545411, j3=110.638538, j4=0.829282, j5=81.75091, j6=11.327332}
  [689] = {j1=-7.14513, j2=-16.545031, j3=110.638266, j4=0.830471, j5=81.751036, j6=11.310935}
  [690] = {j1=-7.1614, j2=-16.544646, j3=110.637991, j4=0.83166, j5=81.751161, j6=11.29454}
  [691] = {j1=-7.177669, j2=-16.544258, j3=110.637713, j4=0.832849, j5=81.751286, j6=11.278145}
  [692] = {j1=-7.193938, j2=-16.543865, j3=110.637433, j4=0.834038, j5=81.75141, j6=11.26175}
  [693] = {j1=-7.210206, j2=-16.543469, j3=110.63715, j4=0.835226, j5=81.751533, j6=11.245357}
  [694] = {j1=-7.226474, j2=-16.543068, j3=110.636864, j4=0.836415, j5=81.751655, j6=11.228964}
  [695] = {j1=-7.24274, j2=-16.542664, j3=110.636575, j4=0.837603, j5=81.751776, j6=11.212572}
  [696] = {j1=-7.259006, j2=-16.542256, j3=110.636283, j4=0.838792, j5=81.751897, j6=11.196181}
  [697] = {j1=-7.275271, j2=-16.541844, j3=110.635989, j4=0.83998, j5=81.752017, j6=11.17979}
  [698] = {j1=-7.291536, j2=-16.541428, j3=110.635691, j4=0.841168, j5=81.752136, j6=11.1634}
  [699] = {j1=-7.307799, j2=-16.541008, j3=110.635391, j4=0.842356, j5=81.752254, j6=11.147011}
  [700] = {j1=-7.324062, j2=-16.540584, j3=110.635088, j4=0.843544, j5=81.752371, j6=11.130622}
  [701] = {j1=-7.340324, j2=-16.540156, j3=110.634782, j4=0.844731, j5=81.752488, j6=11.114234}
  [702] = {j1=-7.356586, j2=-16.539724, j3=110.634474, j4=0.845919, j5=81.752604, j6=11.097847}
  [703] = {j1=-7.372847, j2=-16.539288, j3=110.634162, j4=0.847106, j5=81.752719, j6=11.081461}
  [704] = {j1=-7.389107, j2=-16.538848, j3=110.633848, j4=0.848294, j5=81.752833, j6=11.065075}
  [705] = {j1=-7.405366, j2=-16.538405, j3=110.633531, j4=0.849481, j5=81.752946, j6=11.04869}
  [706] = {j1=-7.421624, j2=-16.537957, j3=110.633211, j4=0.850668, j5=81.753059, j6=11.032306}
  [707] = {j1=-7.437882, j2=-16.537505, j3=110.632888, j4=0.851855, j5=81.753171, j6=11.015923}
  [708] = {j1=-7.454139, j2=-16.53705, j3=110.632563, j4=0.853042, j5=81.753282, j6=10.99954}
  [709] = {j1=-7.470395, j2=-16.53659, j3=110.632234, j4=0.854229, j5=81.753392, j6=10.983159}
  [710] = {j1=-7.486651, j2=-16.536127, j3=110.631903, j4=0.855416, j5=81.753502, j6=10.966777}
  [711] = {j1=-7.502906, j2=-16.53566, j3=110.631569, j4=0.856602, j5=81.75361, j6=10.950397}
  [712] = {j1=-7.51916, j2=-16.535188, j3=110.631232, j4=0.857789, j5=81.753718, j6=10.934017}
  [713] = {j1=-7.535413, j2=-16.534713, j3=110.630893, j4=0.858975, j5=81.753825, j6=10.917639}
  [714] = {j1=-7.551665, j2=-16.534234, j3=110.63055, j4=0.860161, j5=81.753931, j6=10.901261}
  [715] = {j1=-7.567917, j2=-16.533751, j3=110.630205, j4=0.861347, j5=81.754037, j6=10.884883}
  [716] = {j1=-7.584168, j2=-16.533264, j3=110.629857, j4=0.862533, j5=81.754142, j6=10.868507}
  [717] = {j1=-7.600418, j2=-16.532773, j3=110.629506, j4=0.863719, j5=81.754245, j6=10.852131}
  [718] = {j1=-7.616667, j2=-16.532278, j3=110.629152, j4=0.864905, j5=81.754349, j6=10.835756}
  [719] = {j1=-7.632916, j2=-16.531779, j3=110.628795, j4=0.86609, j5=81.754451, j6=10.819382}
  [720] = {j1=-7.649163, j2=-16.531276, j3=110.628436, j4=0.867276, j5=81.754552, j6=10.803008}
  [721] = {j1=-7.66541, j2=-16.530769, j3=110.628074, j4=0.868461, j5=81.754653, j6=10.786636}
  [722] = {j1=-7.681657, j2=-16.530258, j3=110.627709, j4=0.869646, j5=81.754753, j6=10.770264}
  [723] = {j1=-7.697902, j2=-16.529744, j3=110.627341, j4=0.870832, j5=81.754852, j6=10.753893}
  [724] = {j1=-7.714147, j2=-16.529225, j3=110.62697, j4=0.872017, j5=81.75495, j6=10.737522}
  [725] = {j1=-7.73039, j2=-16.528702, j3=110.626597, j4=0.873201, j5=81.755048, j6=10.721153}
  [726] = {j1=-7.746633, j2=-16.528176, j3=110.62622, j4=0.874386, j5=81.755144, j6=10.704784}
  [727] = {j1=-7.762876, j2=-16.527645, j3=110.625841, j4=0.875571, j5=81.75524, j6=10.688416}
  [728] = {j1=-7.779117, j2=-16.527111, j3=110.625459, j4=0.876755, j5=81.755335, j6=10.672049}
  [729] = {j1=-7.795357, j2=-16.526573, j3=110.625074, j4=0.87794, j5=81.75543, j6=10.655683}
  [730] = {j1=-7.811597, j2=-16.52603, j3=110.624687, j4=0.879124, j5=81.755523, j6=10.639317}
  [731] = {j1=-7.827836, j2=-16.525484, j3=110.624296, j4=0.880308, j5=81.755616, j6=10.622952}
  [732] = {j1=-7.844074, j2=-16.524934, j3=110.623903, j4=0.881492, j5=81.755708, j6=10.606589}
  [733] = {j1=-7.860312, j2=-16.52438, j3=110.623507, j4=0.882676, j5=81.755799, j6=10.590225}
  [734] = {j1=-7.876548, j2=-16.523822, j3=110.623108, j4=0.88386, j5=81.755889, j6=10.573863}
  [735] = {j1=-7.892784, j2=-16.52326, j3=110.622706, j4=0.885043, j5=81.755979, j6=10.557502}
  [736] = {j1=-7.909019, j2=-16.522694, j3=110.622302, j4=0.886227, j5=81.756068, j6=10.541141}
  [737] = {j1=-7.925253, j2=-16.522124, j3=110.621894, j4=0.88741, j5=81.756156, j6=10.524781}
  [738] = {j1=-7.941486, j2=-16.52155, j3=110.621484, j4=0.888593, j5=81.756243, j6=10.508422}
  [739] = {j1=-7.957718, j2=-16.520973, j3=110.621071, j4=0.889777, j5=81.756329, j6=10.492064}
  [740] = {j1=-7.97395, j2=-16.520391, j3=110.620655, j4=0.89096, j5=81.756415, j6=10.475707}
  [741] = {j1=-7.990181, j2=-16.519805, j3=110.620237, j4=0.892142, j5=81.7565, j6=10.45935}
  [742] = {j1=-8.00641, j2=-16.519216, j3=110.619815, j4=0.893325, j5=81.756583, j6=10.442994}
  [743] = {j1=-8.022639, j2=-16.518622, j3=110.619391, j4=0.894508, j5=81.756667, j6=10.42664}
  [744] = {j1=-8.038868, j2=-16.518025, j3=110.618964, j4=0.89569, j5=81.756749, j6=10.410286}
  [745] = {j1=-8.055095, j2=-16.517424, j3=110.618534, j4=0.896873, j5=81.756831, j6=10.393932}
  [746] = {j1=-8.071321, j2=-16.516818, j3=110.618101, j4=0.898055, j5=81.756911, j6=10.37758}
  [747] = {j1=-8.087547, j2=-16.516209, j3=110.617665, j4=0.899237, j5=81.756991, j6=10.361229}
  [748] = {j1=-8.103772, j2=-16.515596, j3=110.617227, j4=0.900419, j5=81.757071, j6=10.344878}
  [749] = {j1=-8.119996, j2=-16.514979, j3=110.616786, j4=0.901601, j5=81.757149, j6=10.328528}
  [750] = {j1=-8.136219, j2=-16.514358, j3=110.616342, j4=0.902783, j5=81.757227, j6=10.312179}
  [751] = {j1=-8.152441, j2=-16.513733, j3=110.615895, j4=0.903964, j5=81.757303, j6=10.295831}
  [752] = {j1=-8.168662, j2=-16.513104, j3=110.615445, j4=0.905146, j5=81.757379, j6=10.279484}
  [753] = {j1=-8.184882, j2=-16.512471, j3=110.614993, j4=0.906327, j5=81.757455, j6=10.263138}
  [754] = {j1=-8.201102, j2=-16.511834, j3=110.614537, j4=0.907508, j5=81.757529, j6=10.246792}
  [755] = {j1=-8.217321, j2=-16.511194, j3=110.614079, j4=0.908689, j5=81.757603, j6=10.230447}
  [756] = {j1=-8.233538, j2=-16.510549, j3=110.613618, j4=0.90987, j5=81.757676, j6=10.214104}
  [757] = {j1=-8.249755, j2=-16.5099, j3=110.613154, j4=0.911051, j5=81.757748, j6=10.197761}
  [758] = {j1=-8.265971, j2=-16.509248, j3=110.612688, j4=0.912232, j5=81.757819, j6=10.181419}
  [759] = {j1=-8.282187, j2=-16.508591, j3=110.612218, j4=0.913412, j5=81.757889, j6=10.165078}
  [760] = {j1=-8.298401, j2=-16.507931, j3=110.611746, j4=0.914593, j5=81.757959, j6=10.148737}
  [761] = {j1=-8.314614, j2=-16.507267, j3=110.611271, j4=0.915773, j5=81.758028, j6=10.132398}
  [762] = {j1=-8.330827, j2=-16.506598, j3=110.610793, j4=0.916953, j5=81.758096, j6=10.11606}
  [763] = {j1=-8.347038, j2=-16.505926, j3=110.610312, j4=0.918133, j5=81.758163, j6=10.099722}
  [764] = {j1=-8.363249, j2=-16.50525, j3=110.609829, j4=0.919313, j5=81.75823, j6=10.083385}
  [765] = {j1=-8.379459, j2=-16.50457, j3=110.609342, j4=0.920493, j5=81.758295, j6=10.06705}
  [766] = {j1=-8.395668, j2=-16.503886, j3=110.608853, j4=0.921673, j5=81.75836, j6=10.050715}
  [767] = {j1=-8.411876, j2=-16.503198, j3=110.608361, j4=0.922852, j5=81.758424, j6=10.034381}
  [768] = {j1=-8.428083, j2=-16.502506, j3=110.607866, j4=0.924031, j5=81.758488, j6=10.018047}
  [769] = {j1=-8.444289, j2=-16.50181, j3=110.607369, j4=0.925211, j5=81.75855, j6=10.001715}
  [770] = {j1=-8.460494, j2=-16.501111, j3=110.606868, j4=0.92639, j5=81.758612, j6=9.985384}
  [771] = {j1=-8.476699, j2=-16.500407, j3=110.606365, j4=0.927569, j5=81.758673, j6=9.969054}
  [772] = {j1=-8.492902, j2=-16.499699, j3=110.605859, j4=0.928747, j5=81.758733, j6=9.952724}
  [773] = {j1=-8.509104, j2=-16.498988, j3=110.60535, j4=0.929926, j5=81.758793, j6=9.936395}
  [774] = {j1=-8.525306, j2=-16.498272, j3=110.604838, j4=0.931105, j5=81.758851, j6=9.920068}
  [775] = {j1=-8.541507, j2=-16.497553, j3=110.604323, j4=0.932283, j5=81.758909, j6=9.903741}
  [776] = {j1=-8.557706, j2=-16.49683, j3=110.603806, j4=0.933461, j5=81.758966, j6=9.887415}
  [777] = {j1=-8.573905, j2=-16.496102, j3=110.603286, j4=0.93464, j5=81.759022, j6=9.87109}
  [778] = {j1=-8.590103, j2=-16.495371, j3=110.602763, j4=0.935818, j5=81.759077, j6=9.854766}
  [779] = {j1=-8.6063, j2=-16.494636, j3=110.602237, j4=0.936995, j5=81.759132, j6=9.838443}
  [780] = {j1=-8.622496, j2=-16.493897, j3=110.601708, j4=0.938173, j5=81.759186, j6=9.822121}
  [781] = {j1=-8.638691, j2=-16.493154, j3=110.601177, j4=0.939351, j5=81.759239, j6=9.8058}
  [782] = {j1=-8.654885, j2=-16.492407, j3=110.600642, j4=0.940528, j5=81.759291, j6=9.78948}
  [783] = {j1=-8.671078, j2=-16.491656, j3=110.600105, j4=0.941706, j5=81.759342, j6=9.77316}
  [784] = {j1=-8.68727, j2=-16.490901, j3=110.599565, j4=0.942883, j5=81.759393, j6=9.756842}
  [785] = {j1=-8.703462, j2=-16.490143, j3=110.599022, j4=0.94406, j5=81.759443, j6=9.740525}
  [786] = {j1=-8.719652, j2=-16.48938, j3=110.598477, j4=0.945237, j5=81.759492, j6=9.724208}
  [787] = {j1=-8.735841, j2=-16.488613, j3=110.597928, j4=0.946414, j5=81.75954, j6=9.707893}
  [788] = {j1=-8.75203, j2=-16.487843, j3=110.597377, j4=0.94759, j5=81.759588, j6=9.691578}
  [789] = {j1=-8.768217, j2=-16.487068, j3=110.596823, j4=0.948767, j5=81.759634, j6=9.675264}
  [790] = {j1=-8.784404, j2=-16.48629, j3=110.596266, j4=0.949943, j5=81.75968, j6=9.658952}
  [791] = {j1=-8.800589, j2=-16.485508, j3=110.595706, j4=0.951119, j5=81.759725, j6=9.64264}
  [792] = {j1=-8.816774, j2=-16.484722, j3=110.595144, j4=0.952295, j5=81.75977, j6=9.626329}
  [793] = {j1=-8.832957, j2=-16.483931, j3=110.594578, j4=0.953471, j5=81.759813, j6=9.610019}
  [794] = {j1=-8.84914, j2=-16.483137, j3=110.59401, j4=0.954647, j5=81.759856, j6=9.593711}
  [795] = {j1=-8.865321, j2=-16.482339, j3=110.593439, j4=0.955823, j5=81.759898, j6=9.577403}
  [796] = {j1=-8.881502, j2=-16.481538, j3=110.592865, j4=0.956998, j5=81.759939, j6=9.561096}
  [797] = {j1=-8.897682, j2=-16.480732, j3=110.592289, j4=0.958174, j5=81.759979, j6=9.54479}
  [798] = {j1=-8.91386, j2=-16.479922, j3=110.591709, j4=0.959349, j5=81.760019, j6=9.528485}
  [799] = {j1=-8.930038, j2=-16.479108, j3=110.591127, j4=0.960524, j5=81.760058, j6=9.512181}
  [800] = {j1=-8.946215, j2=-16.478291, j3=110.590542, j4=0.961699, j5=81.760096, j6=9.495878}
  [801] = {j1=-8.96239, j2=-16.477469, j3=110.589954, j4=0.962874, j5=81.760133, j6=9.479576}
  [802] = {j1=-8.978565, j2=-16.476644, j3=110.589363, j4=0.964048, j5=81.760169, j6=9.463275}
  [803] = {j1=-8.994739, j2=-16.475814, j3=110.58877, j4=0.965223, j5=81.760205, j6=9.446975}
  [804] = {j1=-9.010911, j2=-16.474981, j3=110.588173, j4=0.966397, j5=81.76024, j6=9.430676}
  [805] = {j1=-9.027083, j2=-16.474144, j3=110.587574, j4=0.967572, j5=81.760274, j6=9.414378}
  [806] = {j1=-9.043254, j2=-16.473302, j3=110.586972, j4=0.968746, j5=81.760307, j6=9.398081}
  [807] = {j1=-9.059423, j2=-16.472457, j3=110.586367, j4=0.96992, j5=81.760339, j6=9.381785}
  [808] = {j1=-9.075592, j2=-16.471608, j3=110.58576, j4=0.971093, j5=81.760371, j6=9.36549}
  [809] = {j1=-9.09176, j2=-16.470755, j3=110.585149, j4=0.972267, j5=81.760402, j6=9.349196}
  [810] = {j1=-9.107926, j2=-16.469898, j3=110.584536, j4=0.973441, j5=81.760432, j6=9.332903}
  [811] = {j1=-9.124092, j2=-16.469038, j3=110.58392, j4=0.974614, j5=81.760461, j6=9.316611}
  [812] = {j1=-9.140257, j2=-16.468173, j3=110.583301, j4=0.975787, j5=81.76049, j6=9.300319}
  [813] = {j1=-9.15642, j2=-16.467304, j3=110.582679, j4=0.97696, j5=81.760517, j6=9.284029}
  [814] = {j1=-9.172583, j2=-16.466432, j3=110.582054, j4=0.978133, j5=81.760544, j6=9.26774}
  [815] = {j1=-9.188744, j2=-16.465555, j3=110.581427, j4=0.979306, j5=81.76057, j6=9.251452}
  [816] = {j1=-9.204905, j2=-16.464675, j3=110.580797, j4=0.980479, j5=81.760596, j6=9.235166}
  [817] = {j1=-9.221064, j2=-16.46379, j3=110.580164, j4=0.981651, j5=81.76062, j6=9.21888}
  [818] = {j1=-9.237223, j2=-16.462902, j3=110.579528, j4=0.982823, j5=81.760644, j6=9.202595}
  [819] = {j1=-9.25338, j2=-16.46201, j3=110.578889, j4=0.983996, j5=81.760667, j6=9.186311}
  [820] = {j1=-9.269537, j2=-16.461114, j3=110.578248, j4=0.985168, j5=81.760689, j6=9.170028}
  [821] = {j1=-9.285692, j2=-16.460214, j3=110.577603, j4=0.98634, j5=81.760711, j6=9.153746}
  [822] = {j1=-9.301846, j2=-16.45931, j3=110.576956, j4=0.987511, j5=81.760731, j6=9.137465}
  [823] = {j1=-9.317999, j2=-16.458402, j3=110.576306, j4=0.988683, j5=81.760751, j6=9.121186}
  [824] = {j1=-9.334152, j2=-16.45749, j3=110.575653, j4=0.989855, j5=81.76077, j6=9.104907}
  [825] = {j1=-9.350303, j2=-16.456575, j3=110.574998, j4=0.991026, j5=81.760788, j6=9.088629}
  [826] = {j1=-9.366453, j2=-16.455655, j3=110.574339, j4=0.992197, j5=81.760806, j6=9.072353}
  [827] = {j1=-9.382602, j2=-16.454732, j3=110.573678, j4=0.993368, j5=81.760822, j6=9.056077}
  [828] = {j1=-9.39875, j2=-16.453804, j3=110.573014, j4=0.994539, j5=81.760838, j6=9.039802}
  [829] = {j1=-9.414897, j2=-16.452873, j3=110.572347, j4=0.99571, j5=81.760853, j6=9.023529}
  [830] = {j1=-9.431043, j2=-16.451937, j3=110.571677, j4=0.99688, j5=81.760868, j6=9.007257}
  [831] = {j1=-9.447187, j2=-16.450998, j3=110.571005, j4=0.998051, j5=81.760881, j6=8.990985}
  [832] = {j1=-9.463331, j2=-16.450055, j3=110.570329, j4=0.999221, j5=81.760894, j6=8.974715}
  [833] = {j1=-9.479474, j2=-16.449108, j3=110.569651, j4=1.000391, j5=81.760906, j6=8.958446}
  [834] = {j1=-9.495615, j2=-16.448157, j3=110.56897, j4=1.001561, j5=81.760917, j6=8.942177}
  [835] = {j1=-9.511756, j2=-16.447202, j3=110.568286, j4=1.002731, j5=81.760928, j6=8.92591}
  [836] = {j1=-9.527895, j2=-16.446243, j3=110.5676, j4=1.003901, j5=81.760937, j6=8.909644}
  [837] = {j1=-9.544033, j2=-16.445281, j3=110.56691, j4=1.00507, j5=81.760946, j6=8.893379}
  [838] = {j1=-9.560171, j2=-16.444314, j3=110.566218, j4=1.006239, j5=81.760954, j6=8.877116}
  [839] = {j1=-9.576307, j2=-16.443344, j3=110.565523, j4=1.007409, j5=81.760961, j6=8.860853}
  [840] = {j1=-9.592442, j2=-16.442369, j3=110.564825, j4=1.008578, j5=81.760968, j6=8.844591}
  [841] = {j1=-9.608576, j2=-16.441391, j3=110.564124, j4=1.009747, j5=81.760973, j6=8.82833}
  [842] = {j1=-9.624709, j2=-16.440408, j3=110.563421, j4=1.010915, j5=81.760978, j6=8.812071}
  [843] = {j1=-9.64084, j2=-16.439422, j3=110.562714, j4=1.012084, j5=81.760982, j6=8.795812}
  [844] = {j1=-9.656971, j2=-16.438432, j3=110.562005, j4=1.013252, j5=81.760986, j6=8.779555}
  [845] = {j1=-9.673101, j2=-16.437438, j3=110.561293, j4=1.014421, j5=81.760988, j6=8.763299}
  [846] = {j1=-9.689229, j2=-16.43644, j3=110.560578, j4=1.015589, j5=81.76099, j6=8.747043}
  [847] = {j1=-9.705356, j2=-16.435438, j3=110.559861, j4=1.016757, j5=81.760991, j6=8.730789}
  [848] = {j1=-9.721483, j2=-16.434432, j3=110.55914, j4=1.017925, j5=81.760991, j6=8.714536}
  [849] = {j1=-9.737608, j2=-16.433423, j3=110.558417, j4=1.019092, j5=81.760991, j6=8.698284}
  [850] = {j1=-9.753732, j2=-16.432409, j3=110.557691, j4=1.02026, j5=81.760989, j6=8.682034}
  [851] = {j1=-9.769855, j2=-16.431392, j3=110.556962, j4=1.021427, j5=81.760987, j6=8.665784}
  [852] = {j1=-9.785977, j2=-16.43037, j3=110.55623, j4=1.022595, j5=81.760984, j6=8.649535}
  [853] = {j1=-9.802097, j2=-16.429345, j3=110.555495, j4=1.023762, j5=81.76098, j6=8.633288}
  [854] = {j1=-9.818217, j2=-16.428316, j3=110.554758, j4=1.024929, j5=81.760976, j6=8.617041}
  [855] = {j1=-9.834335, j2=-16.427283, j3=110.554018, j4=1.026095, j5=81.76097, j6=8.600796}
  [856] = {j1=-9.850452, j2=-16.426246, j3=110.553275, j4=1.027262, j5=81.760964, j6=8.584552}
  [857] = {j1=-9.866569, j2=-16.425205, j3=110.552529, j4=1.028428, j5=81.760957, j6=8.568309}
  [858] = {j1=-9.882684, j2=-16.42416, j3=110.55178, j4=1.029595, j5=81.76095, j6=8.552067}
  [859] = {j1=-9.898797, j2=-16.423111, j3=110.551029, j4=1.030761, j5=81.760941, j6=8.535827}
  [860] = {j1=-9.91491, j2=-16.422058, j3=110.550274, j4=1.031927, j5=81.760932, j6=8.519587}
  [861] = {j1=-9.931022, j2=-16.421002, j3=110.549517, j4=1.033093, j5=81.760922, j6=8.503348}
  [862] = {j1=-9.947132, j2=-16.419941, j3=110.548757, j4=1.034258, j5=81.760911, j6=8.487111}
  [863] = {j1=-9.963241, j2=-16.418877, j3=110.547995, j4=1.035424, j5=81.7609, j6=8.470875}
  [864] = {j1=-9.97935, j2=-16.417808, j3=110.547229, j4=1.036589, j5=81.760887, j6=8.45464}
  [865] = {j1=-9.995457, j2=-16.416736, j3=110.546461, j4=1.037754, j5=81.760874, j6=8.438406}
  [866] = {j1=-10.011562, j2=-16.41566, j3=110.545689, j4=1.038919, j5=81.76086, j6=8.422173}
  [867] = {j1=-10.027667, j2=-16.41458, j3=110.544915, j4=1.040084, j5=81.760846, j6=8.405941}
  [868] = {j1=-10.043771, j2=-16.413496, j3=110.544138, j4=1.041249, j5=81.76083, j6=8.389711}
  [869] = {j1=-10.059873, j2=-16.412408, j3=110.543359, j4=1.042413, j5=81.760814, j6=8.373482}
  [870] = {j1=-10.075974, j2=-16.411316, j3=110.542576, j4=1.043578, j5=81.760797, j6=8.357253}
  [871] = {j1=-10.092074, j2=-16.410221, j3=110.541791, j4=1.044742, j5=81.760779, j6=8.341026}
  [872] = {j1=-10.108173, j2=-16.409121, j3=110.541003, j4=1.045906, j5=81.760761, j6=8.3248}
  [873] = {j1=-10.124271, j2=-16.408017, j3=110.540212, j4=1.04707, j5=81.760741, j6=8.308576}
  [874] = {j1=-10.140367, j2=-16.40691, j3=110.539418, j4=1.048234, j5=81.760721, j6=8.292352}
  [875] = {j1=-10.156463, j2=-16.405799, j3=110.538621, j4=1.049397, j5=81.7607, j6=8.27613}
  [876] = {j1=-10.172557, j2=-16.404684, j3=110.537822, j4=1.050561, j5=81.760678, j6=8.259909}
  [877] = {j1=-10.18865, j2=-16.403564, j3=110.53702, j4=1.051724, j5=81.760656, j6=8.243689}
  [878] = {j1=-10.204742, j2=-16.402441, j3=110.536215, j4=1.052887, j5=81.760633, j6=8.22747}
  [879] = {j1=-10.220832, j2=-16.401315, j3=110.535407, j4=1.05405, j5=81.760609, j6=8.211252}
  [880] = {j1=-10.236922, j2=-16.400184, j3=110.534596, j4=1.055213, j5=81.760584, j6=8.195035}
  [881] = {j1=-10.25301, j2=-16.399049, j3=110.533783, j4=1.056375, j5=81.760558, j6=8.17882}
  [882] = {j1=-10.269097, j2=-16.39791, j3=110.532966, j4=1.057538, j5=81.760532, j6=8.162606}
  [883] = {j1=-10.285183, j2=-16.396768, j3=110.532147, j4=1.0587, j5=81.760505, j6=8.146393}
  [884] = {j1=-10.301268, j2=-16.395621, j3=110.531325, j4=1.059862, j5=81.760477, j6=8.130181}
  [885] = {j1=-10.317351, j2=-16.394471, j3=110.5305, j4=1.061024, j5=81.760448, j6=8.113971}
  [886] = {j1=-10.333433, j2=-16.393317, j3=110.529673, j4=1.062186, j5=81.760419, j6=8.097761}
  [887] = {j1=-10.349514, j2=-16.392159, j3=110.528842, j4=1.063348, j5=81.760388, j6=8.081553}
  [888] = {j1=-10.365594, j2=-16.390997, j3=110.528009, j4=1.064509, j5=81.760357, j6=8.065346}
  [889] = {j1=-10.381673, j2=-16.389831, j3=110.527173, j4=1.065671, j5=81.760325, j6=8.04914}
  [890] = {j1=-10.39775, j2=-16.388661, j3=110.526334, j4=1.066832, j5=81.760293, j6=8.032936}
  [891] = {j1=-10.413826, j2=-16.387487, j3=110.525492, j4=1.067993, j5=81.760259, j6=8.016732}
  [892] = {j1=-10.429901, j2=-16.38631, j3=110.524648, j4=1.069153, j5=81.760225, j6=8.00053}
  [893] = {j1=-10.445975, j2=-16.385128, j3=110.5238, j4=1.070314, j5=81.76019, j6=7.984329}
  [894] = {j1=-10.462048, j2=-16.383943, j3=110.52295, j4=1.071475, j5=81.760155, j6=7.968129}
  [895] = {j1=-10.478119, j2=-16.382753, j3=110.522097, j4=1.072635, j5=81.760118, j6=7.951931}
  [896] = {j1=-10.494189, j2=-16.38156, j3=110.521242, j4=1.073795, j5=81.760081, j6=7.935733}
  [897] = {j1=-10.510258, j2=-16.380363, j3=110.520383, j4=1.074955, j5=81.760043, j6=7.919537}
  [898] = {j1=-10.526325, j2=-16.379162, j3=110.519521, j4=1.076115, j5=81.760004, j6=7.903342}
  [899] = {j1=-10.542392, j2=-16.377957, j3=110.518657, j4=1.077275, j5=81.759964, j6=7.887148}
  [900] = {j1=-10.558457, j2=-16.376748, j3=110.51779, j4=1.078434, j5=81.759924, j6=7.870956}
  [901] = {j1=-10.574521, j2=-16.375536, j3=110.51692, j4=1.079593, j5=81.759883, j6=7.854765}
  [902] = {j1=-10.590583, j2=-16.374319, j3=110.516048, j4=1.080753, j5=81.759841, j6=7.838575}
  [903] = {j1=-10.606645, j2=-16.373099, j3=110.515172, j4=1.081912, j5=81.759798, j6=7.822386}
  [904] = {j1=-10.622705, j2=-16.371874, j3=110.514294, j4=1.08307, j5=81.759755, j6=7.806199}
  [905] = {j1=-10.638764, j2=-16.370646, j3=110.513412, j4=1.084229, j5=81.759711, j6=7.790012}
  [906] = {j1=-10.654822, j2=-16.369414, j3=110.512528, j4=1.085388, j5=81.759666, j6=7.773827}
  [907] = {j1=-10.670878, j2=-16.368178, j3=110.511642, j4=1.086546, j5=81.75962, j6=7.757643}
  [908] = {j1=-10.686933, j2=-16.366938, j3=110.510752, j4=1.087704, j5=81.759573, j6=7.741461}
  [909] = {j1=-10.702987, j2=-16.365694, j3=110.50986, j4=1.088862, j5=81.759526, j6=7.72528}
  [910] = {j1=-10.71904, j2=-16.364446, j3=110.508964, j4=1.09002, j5=81.759478, j6=7.709099}
  [911] = {j1=-10.735091, j2=-16.363195, j3=110.508066, j4=1.091177, j5=81.759429, j6=7.692921}
  [912] = {j1=-10.751141, j2=-16.361939, j3=110.507165, j4=1.092335, j5=81.759379, j6=7.676743}
  [913] = {j1=-10.76719, j2=-16.36068, j3=110.506262, j4=1.093492, j5=81.759329, j6=7.660567}
  [914] = {j1=-10.783238, j2=-16.359416, j3=110.505355, j4=1.094649, j5=81.759278, j6=7.644392}
  [915] = {j1=-10.799284, j2=-16.358149, j3=110.504446, j4=1.095806, j5=81.759226, j6=7.628218}
  [916] = {j1=-10.815329, j2=-16.356878, j3=110.503534, j4=1.096963, j5=81.759173, j6=7.612045}
  [917] = {j1=-10.831373, j2=-16.355603, j3=110.502619, j4=1.09812, j5=81.75912, j6=7.595874}
  [918] = {j1=-10.847415, j2=-16.354324, j3=110.501701, j4=1.099276, j5=81.759065, j6=7.579704}
  [919] = {j1=-10.863456, j2=-16.353041, j3=110.50078, j4=1.100432, j5=81.75901, j6=7.563536}
  [920] = {j1=-10.879496, j2=-16.351755, j3=110.499857, j4=1.101588, j5=81.758954, j6=7.547368}
  [921] = {j1=-10.895535, j2=-16.350464, j3=110.49893, j4=1.102744, j5=81.758898, j6=7.531202}
  [922] = {j1=-10.911572, j2=-16.34917, j3=110.498001, j4=1.1039, j5=81.75884, j6=7.515037}
  [923] = {j1=-10.927608, j2=-16.347872, j3=110.497069, j4=1.105056, j5=81.758782, j6=7.498873}
  [924] = {j1=-10.943643, j2=-16.346569, j3=110.496135, j4=1.106211, j5=81.758723, j6=7.482711}
  [925] = {j1=-10.959676, j2=-16.345263, j3=110.495197, j4=1.107366, j5=81.758664, j6=7.46655}
  [926] = {j1=-10.975708, j2=-16.343953, j3=110.494257, j4=1.108522, j5=81.758603, j6=7.45039}
  [927] = {j1=-10.991739, j2=-16.34264, j3=110.493314, j4=1.109676, j5=81.758542, j6=7.434232}
  [928] = {j1=-11.007769, j2=-16.341322, j3=110.492368, j4=1.110831, j5=81.75848, j6=7.418075}
  [929] = {j1=-11.023797, j2=-16.34, j3=110.491419, j4=1.111986, j5=81.758417, j6=7.401919}
  [930] = {j1=-11.039824, j2=-16.338675, j3=110.490467, j4=1.11314, j5=81.758354, j6=7.385764}
  [931] = {j1=-11.055849, j2=-16.337345, j3=110.489513, j4=1.114294, j5=81.75829, j6=7.369611}
  [932] = {j1=-11.071873, j2=-16.336012, j3=110.488556, j4=1.115448, j5=81.758224, j6=7.353459}
  [933] = {j1=-11.087896, j2=-16.334675, j3=110.487596, j4=1.116602, j5=81.758159, j6=7.337309}
  [934] = {j1=-11.103918, j2=-16.333334, j3=110.486633, j4=1.117756, j5=81.758092, j6=7.321159}
  [935] = {j1=-11.119938, j2=-16.331989, j3=110.485667, j4=1.118909, j5=81.758025, j6=7.305011}
  [936] = {j1=-11.135957, j2=-16.33064, j3=110.484698, j4=1.120063, j5=81.757957, j6=7.288865}
  [937] = {j1=-11.151975, j2=-16.329287, j3=110.483727, j4=1.121216, j5=81.757888, j6=7.272719}
  [938] = {j1=-11.167991, j2=-16.327931, j3=110.482753, j4=1.122369, j5=81.757818, j6=7.256575}
  [939] = {j1=-11.184006, j2=-16.32657, j3=110.481776, j4=1.123522, j5=81.757748, j6=7.240432}
  [940] = {j1=-11.20002, j2=-16.325206, j3=110.480796, j4=1.124674, j5=81.757676, j6=7.224291}
  [941] = {j1=-11.216032, j2=-16.323838, j3=110.479813, j4=1.125827, j5=81.757604, j6=7.208151}
  [942] = {j1=-11.232043, j2=-16.322466, j3=110.478828, j4=1.126979, j5=81.757532, j6=7.192012}
  [943] = {j1=-11.248053, j2=-16.32109, j3=110.47784, j4=1.128131, j5=81.757458, j6=7.175874}
  [944] = {j1=-11.264061, j2=-16.31971, j3=110.476849, j4=1.129283, j5=81.757384, j6=7.159738}
  [945] = {j1=-11.280068, j2=-16.318326, j3=110.475855, j4=1.130435, j5=81.757309, j6=7.143604}
  [946] = {j1=-11.296074, j2=-16.316939, j3=110.474858, j4=1.131586, j5=81.757233, j6=7.12747}
  [947] = {j1=-11.312078, j2=-16.315547, j3=110.473859, j4=1.132738, j5=81.757157, j6=7.111338}
  [948] = {j1=-11.328081, j2=-16.314152, j3=110.472856, j4=1.133889, j5=81.757079, j6=7.095207}
  [949] = {j1=-11.344082, j2=-16.312753, j3=110.471851, j4=1.13504, j5=81.757001, j6=7.079078}
  [950] = {j1=-11.360083, j2=-16.31135, j3=110.470843, j4=1.136191, j5=81.756922, j6=7.06295}
  [951] = {j1=-11.376081, j2=-16.309943, j3=110.469832, j4=1.137341, j5=81.756843, j6=7.046823}
  [952] = {j1=-11.392079, j2=-16.308532, j3=110.468819, j4=1.138492, j5=81.756762, j6=7.030697}
  [953] = {j1=-11.408075, j2=-16.307117, j3=110.467802, j4=1.139642, j5=81.756681, j6=7.014573}
  [954] = {j1=-11.42407, j2=-16.305699, j3=110.466783, j4=1.140792, j5=81.756599, j6=6.998451}
  [955] = {j1=-11.440063, j2=-16.304276, j3=110.465761, j4=1.141942, j5=81.756517, j6=6.982329}
  [956] = {j1=-11.456055, j2=-16.30285, j3=110.464736, j4=1.143092, j5=81.756433, j6=6.966209}
  [957] = {j1=-11.472046, j2=-16.301419, j3=110.463708, j4=1.144242, j5=81.756349, j6=6.950091}
  [958] = {j1=-11.488035, j2=-16.299985, j3=110.462678, j4=1.145391, j5=81.756264, j6=6.933974}
  [959] = {j1=-11.504023, j2=-16.298547, j3=110.461645, j4=1.14654, j5=81.756179, j6=6.917858}
  [960] = {j1=-11.520009, j2=-16.297106, j3=110.460608, j4=1.147689, j5=81.756092, j6=6.901743}
  [961] = {j1=-11.535994, j2=-16.29566, j3=110.459569, j4=1.148838, j5=81.756005, j6=6.88563}
  [962] = {j1=-11.551978, j2=-16.29421, j3=110.458528, j4=1.149987, j5=81.755917, j6=6.869518}
  [963] = {j1=-11.56796, j2=-16.292757, j3=110.457483, j4=1.151135, j5=81.755828, j6=6.853408}
  [964] = {j1=-11.583941, j2=-16.2913, j3=110.456436, j4=1.152284, j5=81.755739, j6=6.837299}
  [965] = {j1=-11.599921, j2=-16.289838, j3=110.455385, j4=1.153432, j5=81.755648, j6=6.821191}
  [966] = {j1=-11.615899, j2=-16.288373, j3=110.454332, j4=1.15458, j5=81.755557, j6=6.805085}
  [967] = {j1=-11.631876, j2=-16.286904, j3=110.453276, j4=1.155727, j5=81.755466, j6=6.78898}
  [968] = {j1=-11.647851, j2=-16.285432, j3=110.452218, j4=1.156875, j5=81.755373, j6=6.772877}
  [969] = {j1=-11.663825, j2=-16.283955, j3=110.451156, j4=1.158022, j5=81.75528, j6=6.756775}
  [970] = {j1=-11.679797, j2=-16.282474, j3=110.450092, j4=1.15917, j5=81.755186, j6=6.740674}
  [971] = {j1=-11.695769, j2=-16.28099, j3=110.449025, j4=1.160317, j5=81.755091, j6=6.724575}
  [972] = {j1=-11.711738, j2=-16.279502, j3=110.447955, j4=1.161464, j5=81.754995, j6=6.708477}
  [973] = {j1=-11.727707, j2=-16.27801, j3=110.446882, j4=1.16261, j5=81.754899, j6=6.69238}
  [974] = {j1=-11.743673, j2=-16.276514, j3=110.445807, j4=1.163757, j5=81.754802, j6=6.676285}
  [975] = {j1=-11.759639, j2=-16.275014, j3=110.444728, j4=1.164903, j5=81.754704, j6=6.660191}
  [976] = {j1=-11.775603, j2=-16.27351, j3=110.443647, j4=1.166049, j5=81.754605, j6=6.644099}
  [977] = {j1=-11.791566, j2=-16.272002, j3=110.442563, j4=1.167195, j5=81.754506, j6=6.628008}
  [978] = {j1=-11.807527, j2=-16.270491, j3=110.441476, j4=1.168341, j5=81.754406, j6=6.611919}
  [979] = {j1=-11.823487, j2=-16.268976, j3=110.440386, j4=1.169486, j5=81.754305, j6=6.595831}
  [980] = {j1=-11.839445, j2=-16.267456, j3=110.439294, j4=1.170632, j5=81.754203, j6=6.579744}
  [981] = {j1=-11.855402, j2=-16.265933, j3=110.438199, j4=1.171777, j5=81.754101, j6=6.563659}
  [982] = {j1=-11.871357, j2=-16.264406, j3=110.4371, j4=1.172922, j5=81.753998, j6=6.547575}
  [983] = {j1=-11.887311, j2=-16.262876, j3=110.436, j4=1.174067, j5=81.753894, j6=6.531493}
  [984] = {j1=-11.903264, j2=-16.261341, j3=110.434896, j4=1.175211, j5=81.753789, j6=6.515412}
  [985] = {j1=-11.919215, j2=-16.259803, j3=110.433789, j4=1.176356, j5=81.753684, j6=6.499332}
  [986] = {j1=-11.935165, j2=-16.25826, j3=110.43268, j4=1.1775, j5=81.753578, j6=6.483254}
  [987] = {j1=-11.951113, j2=-16.256714, j3=110.431568, j4=1.178644, j5=81.753471, j6=6.467177}
  [988] = {j1=-11.96706, j2=-16.255164, j3=110.430453, j4=1.179788, j5=81.753363, j6=6.451102}
  [989] = {j1=-11.983005, j2=-16.25361, j3=110.429335, j4=1.180932, j5=81.753254, j6=6.435028}
  [990] = {j1=-11.998949, j2=-16.252052, j3=110.428214, j4=1.182075, j5=81.753145, j6=6.418956}
  [991] = {j1=-12.014892, j2=-16.250491, j3=110.427091, j4=1.183219, j5=81.753035, j6=6.402885}
  [992] = {j1=-12.030833, j2=-16.248925, j3=110.425964, j4=1.184362, j5=81.752925, j6=6.386816}
  [993] = {j1=-12.046772, j2=-16.247356, j3=110.424835, j4=1.185505, j5=81.752813, j6=6.370748}
  [994] = {j1=-12.06271, j2=-16.245782, j3=110.423703, j4=1.186647, j5=81.752701, j6=6.354681}
  [995] = {j1=-12.078647, j2=-16.244205, j3=110.422569, j4=1.18779, j5=81.752588, j6=6.338616}
  [996] = {j1=-12.094582, j2=-16.242624, j3=110.421431, j4=1.188932, j5=81.752474, j6=6.322552}
  [997] = {j1=-12.110516, j2=-16.24104, j3=110.420291, j4=1.190074, j5=81.75236, j6=6.30649}
  [998] = {j1=-12.126448, j2=-16.239451, j3=110.419148, j4=1.191216, j5=81.752245, j6=6.290429}
  [999] = {j1=-12.142379, j2=-16.237859, j3=110.418002, j4=1.192358, j5=81.752129, j6=6.27437}
public pointRx pCad[1000]
  [0] = {rx=0.301954, ry=175.773713, rz=18.532164, fatherId=world[0]}
  [1] = {y=-0.146773, rx=0.301951, ry=175.773713, rz=18.532167, fatherId=world[0]}
  [2] = {y=-0.293546, rx=0.301948, ry=175.773713, rz=18.53217, fatherId=world[0]}
  [3] = {y=-0.440319, rx=0.301945, ry=175.773712, rz=18.532173, fatherId=world[0]}
  [4] = {y=-0.587091, rx=0.301942, ry=175.773712, rz=18.532176, fatherId=world[0]}
  [5] = {y=-0.733864, rx=0.301938, ry=175.773712, rz=18.53218, fatherId=world[0]}
  [6] = {y=-0.880637, rx=0.301935, ry=175.773711, rz=18.532183, fatherId=world[0]}
  [7] = {y=-1.02741, rx=0.301932, ry=175.773711, rz=18.532186, fatherId=world[0]}
  [8] = {x=-1E-06, y=-1.174183, rx=0.301929, ry=175.773711, rz=18.532189, fatherId=world[0]}
  [9] = {x=-1E-06, y=-1.320956, rx=0.301926, ry=175.77371, rz=18.532192, fatherId=world[0]}
  [10] = {x=-1E-06, y=-1.467729, rx=0.301922, ry=175.77371, rz=18.532196, fatherId=world[0]}
  [11] = {x=-1E-06, y=-1.614501, rx=0.301919, ry=175.77371, rz=18.532199, fatherId=world[0]}
  [12] = {x=-1E-06, y=-1.761274, rx=0.301916, ry=175.773709, rz=18.532202, fatherId=world[0]}
  [13] = {x=-1E-06, y=-1.908047, rx=0.301913, ry=175.773709, rz=18.532205, fatherId=world[0]}
  [14] = {x=-1E-06, y=-2.05482, rx=0.30191, ry=175.773709, rz=18.532208, fatherId=world[0]}
  [15] = {x=-1E-06, y=-2.201593, rx=0.301906, ry=175.773708, rz=18.532211, fatherId=world[0]}
  [16] = {x=-1E-06, y=-2.348366, rx=0.301903, ry=175.773708, rz=18.532215, fatherId=world[0]}
  [17] = {x=-1E-06, y=-2.495139, rx=0.3019, ry=175.773708, rz=18.532218, fatherId=world[0]}
  [18] = {x=-1E-06, y=-2.641911, rx=0.301897, ry=175.773707, rz=18.532221, fatherId=world[0]}
  [19] = {x=-1E-06, y=-2.788684, rx=0.301894, ry=175.773707, rz=18.532224, fatherId=world[0]}
  [20] = {x=-1E-06, y=-2.935457, rx=0.30189, ry=175.773707, rz=18.532227, fatherId=world[0]}
  [21] = {x=-1E-06, y=-3.08223, rx=0.301887, ry=175.773706, rz=18.532231, fatherId=world[0]}
  [22] = {x=-1E-06, y=-3.229003, rx=0.301884, ry=175.773706, rz=18.532234, fatherId=world[0]}
  [23] = {x=-1E-06, y=-3.375776, rx=0.301881, ry=175.773706, rz=18.532237, fatherId=world[0]}
  [24] = {x=-2E-06, y=-3.522549, rx=0.301878, ry=175.773705, rz=18.53224, fatherId=world[0]}
  [25] = {x=-2E-06, y=-3.669321, rx=0.301874, ry=175.773705, rz=18.532243, fatherId=world[0]}
  [26] = {x=-2E-06, y=-3.816094, rx=0.301871, ry=175.773705, rz=18.532246, fatherId=world[0]}
  [27] = {x=-2E-06, y=-3.962867, rx=0.301868, ry=175.773705, rz=18.53225, fatherId=world[0]}
  [28] = {x=-2E-06, y=-4.10964, rx=0.301865, ry=175.773704, rz=18.532253, fatherId=world[0]}
  [29] = {x=-2E-06, y=-4.256413, rx=0.301862, ry=175.773704, rz=18.532256, fatherId=world[0]}
  [30] = {x=-2E-06, y=-4.403186, rx=0.301859, ry=175.773704, rz=18.532259, fatherId=world[0]}
  [31] = {x=-2E-06, y=-4.549959, rx=0.301855, ry=175.773703, rz=18.532262, fatherId=world[0]}
  [32] = {x=-2E-06, y=-4.696731, rx=0.301852, ry=175.773703, rz=18.532266, fatherId=world[0]}
  [33] = {x=-2E-06, y=-4.843504, rx=0.301849, ry=175.773703, rz=18.532269, fatherId=world[0]}
  [34] = {x=-2E-06, y=-4.990277, rx=0.301846, ry=175.773702, rz=18.532272, fatherId=world[0]}
  [35] = {x=-2E-06, y=-5.13705, rx=0.301843, ry=175.773702, rz=18.532275, fatherId=world[0]}
  [36] = {x=-2E-06, y=-5.283823, rx=0.301839, ry=175.773702, rz=18.532278, fatherId=world[0]}
  [37] = {x=-2E-06, y=-5.430596, rx=0.301836, ry=175.773701, rz=18.532281, fatherId=world[0]}
  [38] = {x=-2E-06, y=-5.577369, rx=0.301833, ry=175.773701, rz=18.532285, fatherId=world[0]}
  [39] = {x=-3E-06, y=-5.724141, rx=0.30183, ry=175.773701, rz=18.532288, fatherId=world[0]}
  [40] = {x=-3E-06, y=-5.870914, rx=0.301827, ry=175.773701, rz=18.532291, fatherId=world[0]}
  [41] = {x=-3E-06, y=-6.017687, rx=0.301823, ry=175.7737, rz=18.532294, fatherId=world[0]}
  [42] = {x=-3E-06, y=-6.16446, rx=0.30182, ry=175.7737, rz=18.532297, fatherId=world[0]}
  [43] = {x=-3E-06, y=-6.311233, rx=0.301817, ry=175.7737, rz=18.532301, fatherId=world[0]}
  [44] = {x=-3E-06, y=-6.458006, rx=0.301814, ry=175.773699, rz=18.532304, fatherId=world[0]}
  [45] = {x=-3E-06, y=-6.604779, rx=0.301811, ry=175.773699, rz=18.532307, fatherId=world[0]}
  [46] = {x=-3E-06, y=-6.751551, rx=0.301807, ry=175.773699, rz=18.53231, fatherId=world[0]}
  [47] = {x=-3E-06, y=-6.898324, rx=0.301804, ry=175.773698, rz=18.532313, fatherId=world[0]}
  [48] = {x=-3E-06, y=-7.045097, rx=0.301801, ry=175.773698, rz=18.532317, fatherId=world[0]}
  [49] = {x=-3E-06, y=-7.19187, rx=0.301798, ry=175.773698, rz=18.53232, fatherId=world[0]}
  [50] = {x=-3E-06, y=-7.338643, rx=0.301795, ry=175.773698, rz=18.532323, fatherId=world[0]}
  [51] = {x=-3E-06, y=-7.485416, rx=0.301791, ry=175.773697, rz=18.532326, fatherId=world[0]}
  [52] = {x=-3E-06, y=-7.632189, rx=0.301788, ry=175.773697, rz=18.532329, fatherId=world[0]}
  [53] = {x=-3E-06, y=-7.778961, rx=0.301785, ry=175.773697, rz=18.532332, fatherId=world[0]}
  [54] = {x=-4E-06, y=-7.925734, rx=0.301782, ry=175.773696, rz=18.532336, fatherId=world[0]}
